LIN {X 0,Y 612.539,Z 280.742,A -85,B 0,C 180,E1 -8059.322,E2 -8059.322} C_VEL
LIN {X 0,Y 612.53,Z 280.74,A -85,B 0,C 180,E1 -8062.097,E2 -8062.097} C_VEL
LIN {X 0,Y 612.605,Z 280.734,A -85,B 0,C 180,E1 -8064.329,E2 -8064.329} C_VEL
LIN {X 0,Y 612.556,Z 280.744,A -85,B 0,C 180,E1 -8066.71,E2 -8066.71} C_VEL
LIN {X 0,Y 612.575,Z 280.737,A -85,B 0,C 180,E1 -8069.048,E2 -8069.048} C_VEL
LIN {X 0,Y 612.575,Z 280.734,A -85,B 0,C 180,E1 -8071.698,E2 -8071.698} C_VEL
LIN {X 0,Y 612.557,Z 280.743,A -85,B 0,C 180,E1 -8074.603,E2 -8074.603} C_VEL
LIN {X 0,Y 612.586,Z 280.736,A -85,B 0,C 180,E1 -8077.122,E2 -8077.122} C_VEL
LIN {X 0,Y 612.607,Z 280.742,A -85,B 0,C 180,E1 -8079.939,E2 -8079.939} C_VEL
LIN {X 0,Y 612.586,Z 280.735,A -85,B 0,C 180,E1 -8082.705,E2 -8082.705} C_VEL
LIN {X 0,Y 612.61,Z 280.735,A -85,B 0,C 180,E1 -8085.431,E2 -8085.431} C_VEL
LIN {X 0,Y 612.595,Z 280.739,A -85,B 0,C 180,E1 -8087.453,E2 -8087.453} C_VEL
LIN {X 0,Y 612.647,Z 280.829,A -85,B 0,C 180,E1 -8088.751,E2 -8088.751} C_VEL
LIN {X 0,Y 614.455,Z 290.422,A -85,B 0,C 180,E1 -8089.989,E2 -8089.989} C_VEL
LIN {X 0,Y 614.314,Z 310.578,A -85,B 0,C 180,E1 -8092.465,E2 -8092.465} C_VEL
LIN {X 0,Y 613.746,Z 335.947,A -85,B 0,C 180,E1 -8095.582,E2 -8095.582} C_VEL
LIN {X 0,Y 613.659,Z 342.221,A -85,B 0,C 180,E1 -8096.36,E2 -8096.36} C_VEL
LIN {X 0,Y 616.099,Z 357.034,A -85,B 0,C 180,E1 -8096.639,E2 -8096.639} C_VEL
LIN {X 0,Y 614.848,Z 480.497,A -85,B 0,C 180,E1 -8098.246,E2 -8098.246} C_VEL
LIN {X 0,Y 614.62,Z 495.222,A -85,B 0,C 180,E1 -8098.571,E2 -8098.571} C_VEL
LIN {X 0,Y 614.253,Z 509.138,A -85,B 0,C 180,E1 -8099.02,E2 -8099.02} C_VEL
LIN {X 0,Y 613.913,Z 520.829,A -85,B 0,C 180,E1 -8099.51,E2 -8099.51} C_VEL
LIN {X 0,Y 613.489,Z 533.262,A -85,B 0,C 180,E1 -8100.164,E2 -8100.164} C_VEL
LIN {X 0,Y 613.212,Z 545.749,A -85,B 0,C 180,E1 -8100.982,E2 -8100.982} C_VEL
LIN {X 0,Y 612.816,Z 556.08,A -85,B 0,C 180,E1 -8101.801,E2 -8101.801} C_VEL
LIN {X 0,Y 612.393,Z 566.382,A -85,B 0,C 180,E1 -8102.786,E2 -8102.786} C_VEL
LIN {X 0,Y 612.12,Z 574.899,A -85,B 0,C 180,E1 -8103.773,E2 -8103.773} C_VEL
LIN {X 0,Y 611.915,Z 583.24,A -85,B 0,C 180,E1 -8104.95,E2 -8104.95} C_VEL
LIN {X 0,Y 611.86,Z 588.773,A -85,B 0,C 180,E1 -8105.914,E2 -8105.914} C_VEL
LIN {X 0,Y 611.734,Z 593.465,A -85,B 0,C 180,E1 -8106.905,E2 -8106.905} C_VEL
LIN {X 0,Y 611.594,Z 598.317,A -85,B 0,C 180,E1 -8108.231,E2 -8108.231} C_VEL
LIN {X 0,Y 611.56,Z 600.925,A -85,B 0,C 180,E1 -8109.227,E2 -8109.227} C_VEL
LIN {X 0,Y 611.605,Z 602.329,A -85,B 0,C 180,E1 -8109.959,E2 -8109.959} C_VEL
LIN {X 0,Y 611.466,Z 603.754,A -85,B 0,C 180,E1 -8111.229,E2 -8111.229} C_VEL
LIN {X 0,Y 611.5,Z 603.889,A -85,B 0,C 180,E1 -8112.57,E2 -8112.57} C_VEL
LIN {X 0,Y 611.564,Z 603.427,A -85,B 0,C 180,E1 -8113.242,E2 -8113.242} C_VEL
LIN {X 0,Y 611.514,Z 601.388,A -85,B 0,C 180,E1 -8114.596,E2 -8114.596} C_VEL
LIN {X 0,Y 611.62,Z 597.836,A -85,B 0,C 180,E1 -8115.953,E2 -8115.953} C_VEL
LIN {X 0,Y 611.67,Z 594.126,A -85,B 0,C 180,E1 -8116.978,E2 -8116.978} C_VEL
LIN {X 0,Y 611.798,Z 588.668,A -85,B 0,C 180,E1 -8118.144,E2 -8118.144} C_VEL
LIN {X 0,Y 611.995,Z 581.268,A -85,B 0,C 180,E1 -8119.385,E2 -8119.385} C_VEL
LIN {X 0,Y 612.218,Z 573.296,A -85,B 0,C 180,E1 -8120.464,E2 -8120.464} C_VEL
LIN {X 0,Y 612.47,Z 564.315,A -85,B 0,C 180,E1 -8121.467,E2 -8121.467} C_VEL
LIN {X 0,Y 612.872,Z 553.36,A -85,B 0,C 180,E1 -8122.476,E2 -8122.476} C_VEL
LIN {X 0,Y 613.238,Z 542.494,A -85,B 0,C 180,E1 -8123.296,E2 -8123.296} C_VEL
LIN {X 0,Y 613.619,Z 530.354,A -85,B 0,C 180,E1 -8124.047,E2 -8124.047} C_VEL
LIN {X 0,Y 613.943,Z 517.245,A -85,B 0,C 180,E1 -8124.699,E2 -8124.699} C_VEL
LIN {X 0,Y 614.354,Z 503.666,A -85,B 0,C 180,E1 -8125.222,E2 -8125.222} C_VEL
LIN {X 0,Y 614.635,Z 489.847,A -85,B 0,C 180,E1 -8125.616,E2 -8125.616} C_VEL
LIN {X 0,Y 614.816,Z 476.132,A -85,B 0,C 180,E1 -8125.88,E2 -8125.88} C_VEL
LIN {X 0,Y 615.787,Z 356.431,A -85,B 0,C 180,E1 -8127.383,E2 -8127.383} C_VEL
LIN {X 0,Y 613.434,Z 341.628,A -85,B 0,C 180,E1 -8127.642,E2 -8127.642} C_VEL
LIN {X 0,Y 613.881,Z 320.293,A -85,B 0,C 180,E1 -8130.325,E2 -8130.325} C_VEL
LIN {X 0,Y 614.329,Z 299.291,A -85,B 0,C 180,E1 -8132.967,E2 -8132.967} C_VEL
LIN {X 0,Y 614.456,Z 291.433,A -85,B 0,C 180,E1 -8133.957,E2 -8133.957} C_VEL
LIN {X 0,Y 612.592,Z 280.737,A -85,B 0,C 180,E1 -8135.395,E2 -8135.395} C_VEL
LIN {X 0,Y 612.548,Z 280.745,A -85,B 0,C 180,E1 -8138.133,E2 -8138.133} C_VEL
LIN {X 0,Y 612.54,Z 280.738,A -85,B 0,C 180,E1 -8140.998,E2 -8140.998} C_VEL
LIN {X 0,Y 612.553,Z 280.742,A -85,B 0,C 180,E1 -8143.912,E2 -8143.912} C_VEL
LIN {X 0,Y 612.551,Z 280.743,A -85,B 0,C 180,E1 -8144.184,E2 -8144.184} C_VEL
LIN {X 0,Y 611.899,Z 280.825,A -85,B 0,C 180,E1 -8144.733,E2 -8144.733} C_VEL
LIN {X 0,Y 609.053,Z 281.178,A -85,B 0,C 180,E1 -8145.624,E2 -8145.624} C_VEL
LIN {X 0,Y 606.631,Z 281.478,A -85,B 0,C 180,E1 -8146.34,E2 -8146.34} C_VEL
LIN {X 0,Y 605.577,Z 281.607,A -85,B 0,C 180,E1 -8146.893,E2 -8146.893} C_VEL
LIN {X 0,Y 605.485,Z 281.618,A -85,B 0,C 180,E1 -8147.08,E2 -8147.08} C_VEL
LIN {X 0,Y 605.499,Z 281.622,A -85,B 0,C 180,E1 -8149.773,E2 -8149.773} C_VEL
LIN {X 0,Y 605.482,Z 281.62,A -85,B 0,C 180,E1 -8152.183,E2 -8152.183} C_VEL
LIN {X 0,Y 605.512,Z 281.616,A -85,B 0,C 180,E1 -8154.661,E2 -8154.661} C_VEL
LIN {X 0,Y 605.519,Z 281.619,A -85,B 0,C 180,E1 -8157.612,E2 -8157.612} C_VEL
LIN {X 0,Y 605.509,Z 281.616,A -85,B 0,C 180,E1 -8160.18,E2 -8160.18} C_VEL
LIN {X 0,Y 605.497,Z 281.62,A -85,B 0,C 180,E1 -8162.436,E2 -8162.436} C_VEL
LIN {X 0,Y 605.528,Z 281.615,A -85,B 0,C 180,E1 -8165.389,E2 -8165.389} C_VEL
LIN {X 0,Y 605.548,Z 281.615,A -85,B 0,C 180,E1 -8168.274,E2 -8168.274} C_VEL
LIN {X 0,Y 605.564,Z 281.61,A -85,B 0,C 180,E1 -8171.101,E2 -8171.101} C_VEL
LIN {X 0,Y 605.58,Z 281.609,A -85,B 0,C 180,E1 -8173.882,E2 -8173.882} C_VEL
LIN {X 0,Y 605.61,Z 281.604,A -85,B 0,C 180,E1 -8176.624,E2 -8176.624} C_VEL
LIN {X 0,Y 605.595,Z 281.605,A -85,B 0,C 180,E1 -8179.46,E2 -8179.46} C_VEL
LIN {X 0,Y 605.638,Z 281.602,A -85,B 0,C 180,E1 -8182.69,E2 -8182.69} C_VEL
LIN {X 0,Y 605.665,Z 281.693,A -85,B 0,C 180,E1 -8183.534,E2 -8183.534} C_VEL
LIN {X 0,Y 606.536,Z 288.286,A -85,B 0,C 180,E1 -8184.698,E2 -8184.698} C_VEL
LIN {X 0,Y 606.366,Z 297.794,A -85,B 0,C 180,E1 -8186.314,E2 -8186.314} C_VEL
LIN {X 0,Y 609.016,Z 310.551,A -85,B 0,C 180,E1 -8186.537,E2 -8186.537} C_VEL
LIN {X 0,Y 608.253,Z 432.958,A -85,B 0,C 180,E1 -8187.998,E2 -8187.998} C_VEL
LIN {X 0,Y 608.073,Z 447.42,A -85,B 0,C 180,E1 -8188.307,E2 -8188.307} C_VEL
LIN {X 0,Y 607.806,Z 460.691,A -85,B 0,C 180,E1 -8188.719,E2 -8188.719} C_VEL
LIN {X 0,Y 607.447,Z 473.678,A -85,B 0,C 180,E1 -8189.255,E2 -8189.255} C_VEL
LIN {X 0,Y 607.1,Z 486.217,A -85,B 0,C 180,E1 -8189.916,E2 -8189.916} C_VEL
LIN {X 0,Y 606.605,Z 497.697,A -85,B 0,C 180,E1 -8190.66,E2 -8190.66} C_VEL
LIN {X 0,Y 606.277,Z 508.19,A -85,B 0,C 180,E1 -8191.488,E2 -8191.488} C_VEL
LIN {X 0,Y 605.795,Z 518.648,A -85,B 0,C 180,E1 -8192.483,E2 -8192.483} C_VEL
LIN {X 0,Y 605.512,Z 527.271,A -85,B 0,C 180,E1 -8193.48,E2 -8193.48} C_VEL
LIN {X 0,Y 605.174,Z 534.48,A -85,B 0,C 180,E1 -8194.479,E2 -8194.479} C_VEL
LIN {X 0,Y 605.072,Z 541.182,A -85,B 0,C 180,E1 -8195.612,E2 -8195.612} C_VEL
LIN {X 0,Y 604.868,Z 546.167,A -85,B 0,C 180,E1 -8196.648,E2 -8196.648} C_VEL
LIN {X 0,Y 604.685,Z 551.137,A -85,B 0,C 180,E1 -8197.988,E2 -8197.988} C_VEL
LIN {X 0,Y 604.615,Z 554.619,A -85,B 0,C 180,E1 -8199.332,E2 -8199.332} C_VEL
LIN {X 0,Y 604.562,Z 556.716,A -85,B 0,C 180,E1 -8200.681,E2 -8200.681} C_VEL
LIN {X 0,Y 604.528,Z 557.462,A -85,B 0,C 180,E1 -8202.036,E2 -8202.036} C_VEL
LIN {X 0,Y 604.611,Z 556.839,A -85,B 0,C 180,E1 -8203.395,E2 -8203.395} C_VEL
LIN {X 0,Y 604.618,Z 554.819,A -85,B 0,C 180,E1 -8204.764,E2 -8204.764} C_VEL
LIN {X 0,Y 604.762,Z 551.338,A -85,B 0,C 180,E1 -8206.137,E2 -8206.137} C_VEL
LIN {X 0,Y 604.901,Z 546.275,A -85,B 0,C 180,E1 -8207.52,E2 -8207.52} C_VEL
LIN {X 0,Y 605.11,Z 541.411,A -85,B 0,C 180,E1 -8208.541,E2 -8208.541} C_VEL
LIN {X 0,Y 605.398,Z 534.08,A -85,B 0,C 180,E1 -8209.779,E2 -8209.779} C_VEL
LIN {X 0,Y 605.675,Z 526.294,A -85,B 0,C 180,E1 -8210.845,E2 -8210.845} C_VEL
LIN {X 0,Y 606.124,Z 517.12,A -85,B 0,C 180,E1 -8211.879,E2 -8211.879} C_VEL
LIN {X 0,Y 606.513,Z 507.043,A -85,B 0,C 180,E1 -8212.821,E2 -8212.821} C_VEL
LIN {X 0,Y 607.008,Z 495.237,A -85,B 0,C 180,E1 -8213.728,E2 -8213.728} C_VEL
LIN {X 0,Y 607.408,Z 483.868,A -85,B 0,C 180,E1 -8214.44,E2 -8214.44} C_VEL
LIN {X 0,Y 607.866,Z 470.729,A -85,B 0,C 180,E1 -8215.097,E2 -8215.097} C_VEL
LIN {X 0,Y 608.202,Z 456.909,A -85,B 0,C 180,E1 -8215.63,E2 -8215.63} C_VEL
LIN {X 0,Y 608.475,Z 441.955,A -85,B 0,C 180,E1 -8216.045,E2 -8216.045} C_VEL
LIN {X 0,Y 608.6,Z 428.129,A -85,B 0,C 180,E1 -8216.291,E2 -8216.291} C_VEL
LIN {X 0,Y 609.415,Z 310.991,A -85,B 0,C 180,E1 -8217.691,E2 -8217.691} C_VEL
LIN {X 0,Y 606.657,Z 298.091,A -85,B 0,C 180,E1 -8217.943,E2 -8217.943} C_VEL
LIN {X 0,Y 606.757,Z 288.755,A -85,B 0,C 180,E1 -8219.569,E2 -8219.569} C_VEL
LIN {X 0,Y 605.499,Z 281.623,A -85,B 0,C 180,E1 -8220.897,E2 -8220.897} C_VEL
LIN {X 0,Y 605.495,Z 281.62,A -85,B 0,C 180,E1 -8223.727,E2 -8223.727} C_VEL
LIN {X 0,Y 605.501,Z 281.623,A -85,B 0,C 180,E1 -8226.152,E2 -8226.152} C_VEL
LIN {X 0,Y 605.486,Z 281.616,A -85,B 0,C 180,E1 -8229.188,E2 -8229.188} C_VEL
LIN {X 0,Y 605.471,Z 281.624,A -85,B 0,C 180,E1 -8232.14,E2 -8232.14} C_VEL
LIN {X 0,Y 605.489,Z 281.609,A -85,B 0,C 180,E1 -8234.88,E2 -8234.88} C_VEL
LIN {X 0,Y 605.48,Z 281.624,A -85,B 0,C 180,E1 -8237.858,E2 -8237.858} C_VEL
LIN {X 0,Y 605.487,Z 281.617,A -85,B 0,C 180,E1 -8240.487,E2 -8240.487} C_VEL
LIN {X 0,Y 605.524,Z 281.609,A -85,B 0,C 180,E1 -8243.022,E2 -8243.022} C_VEL
LIN {X 0,Y 605.481,Z 281.611,A -85,B 0,C 180,E1 -8245.469,E2 -8245.469} C_VEL
LIN {X 0,Y 605.492,Z 281.622,A -85,B 0,C 180,E1 -8247.85,E2 -8247.85} C_VEL
LIN {X 0,Y 605.528,Z 281.614,A -85,B 0,C 180,E1 -8250.172,E2 -8250.172} C_VEL
LIN {X 0,Y 605.487,Z 281.612,A -85,B 0,C 180,E1 -8252.437,E2 -8252.437} C_VEL
LIN {X 0,Y 605.509,Z 281.62,A -85,B 0,C 180,E1 -8255.39,E2 -8255.39} C_VEL
LIN {X 0,Y 605.53,Z 281.618,A -85,B 0,C 180,E1 -8257.722,E2 -8257.722} C_VEL
LIN {X 0,Y 605.527,Z 281.608,A -85,B 0,C 180,E1 -8260.4,E2 -8260.4} C_VEL
LIN {X 0,Y 605.517,Z 281.617,A -85,B 0,C 180,E1 -8263.19,E2 -8263.19} C_VEL
LIN {X 0,Y 605.567,Z 281.603,A -85,B 0,C 180,E1 -8265.942,E2 -8265.942} C_VEL
LIN {X 0,Y 605.545,Z 281.609,A -85,B 0,C 180,E1 -8268.659,E2 -8268.659} C_VEL
LIN {X 0,Y 605.533,Z 281.608,A -85,B 0,C 180,E1 -8270.68,E2 -8270.68} C_VEL
LIN {X 0,Y 605.638,Z 281.605,A -85,B 0,C 180,E1 -8273.359,E2 -8273.359} C_VEL
LIN {X 0,Y 605.651,Z 281.589,A -85,B 0,C 180,E1 -8276.021,E2 -8276.021} C_VEL
LIN {X 0,Y 605.776,Z 281.585,A -85,B 0,C 180,E1 -8279.338,E2 -8279.338} C_VEL
LIN {X 0,Y 605.781,Z 281.578,A -85,B 0,C 180,E1 -8281.325,E2 -8281.325} C_VEL
LIN {X 0,Y 605.666,Z 281.597,A -85,B 0,C 180,E1 -8284.643,E2 -8284.643} C_VEL
LIN {X 0,Y 605.616,Z 281.598,A -85,B 0,C 180,E1 -8287.309,E2 -8287.309} C_VEL
LIN {X 0,Y 605.635,Z 281.602,A -85,B 0,C 180,E1 -8290.664,E2 -8290.664} C_VEL
LIN {X 0,Y 605.588,Z 281.6,A -85,B 0,C 180,E1 -8293.705,E2 -8293.705} C_VEL
LIN {X 0,Y 605.543,Z 281.611,A -85,B 0,C 180,E1 -8296.809,E2 -8296.809} C_VEL
LIN {X 0,Y 605.543,Z 281.615,A -85,B 0,C 180,E1 -8298.898,E2 -8298.898} C_VEL
LIN {X 0,Y 605.519,Z 281.607,A -85,B 0,C 180,E1 -8301.726,E2 -8301.726} C_VEL
LIN {X 0,Y 605.523,Z 281.611,A -85,B 0,C 180,E1 -8303.965,E2 -8303.965} C_VEL
LIN {X 0,Y 605.476,Z 281.622,A -85,B 0,C 180,E1 -8306.819,E2 -8306.819} C_VEL
LIN {X 0,Y 605.529,Z 281.612,A -85,B 0,C 180,E1 -8309.067,E2 -8309.067} C_VEL
LIN {X 0,Y 605.536,Z 281.609,A -85,B 0,C 180,E1 -8311.368,E2 -8311.368} C_VEL
LIN {X 0,Y 605.514,Z 281.608,A -85,B 0,C 180,E1 -8314.529,E2 -8314.529} C_VEL
LIN {X 0,Y 605.549,Z 281.606,A -85,B 0,C 180,E1 -8317.052,E2 -8317.052} C_VEL
LIN {X 0,Y 605.509,Z 281.613,A -85,B 0,C 180,E1 -8319.512,E2 -8319.512} C_VEL
LIN {X 0,Y 605.507,Z 281.621,A -85,B 0,C 180,E1 -8322.243,E2 -8322.243} C_VEL
LIN {X 0,Y 605.499,Z 281.613,A -85,B 0,C 180,E1 -8325.121,E2 -8325.121} C_VEL
LIN {X 0,Y 605.53,Z 281.615,A -85,B 0,C 180,E1 -8327.866,E2 -8327.866} C_VEL
LIN {X 0,Y 605.514,Z 281.617,A -85,B 0,C 180,E1 -8330.492,E2 -8330.492} C_VEL
LIN {X 0,Y 605.581,Z 281.604,A -85,B 0,C 180,E1 -8333.028,E2 -8333.028} C_VEL
LIN {X 0,Y 605.519,Z 281.619,A -85,B 0,C 180,E1 -8335.474,E2 -8335.474} C_VEL
LIN {X 0,Y 605.51,Z 281.626,A -85,B 0,C 180,E1 -8337.854,E2 -8337.854} C_VEL
LIN {X 0,Y 605.54,Z 281.619,A -85,B 0,C 180,E1 -8340.175,E2 -8340.175} C_VEL
LIN {X 0,Y 605.504,Z 281.62,A -85,B 0,C 180,E1 -8342.44,E2 -8342.44} C_VEL
LIN {X 0,Y 605.53,Z 281.746,A -85,B 0,C 180,E1 -8343.857,E2 -8343.857} C_VEL
LIN {X 0,Y 608.272,Z 294.613,A -85,B 0,C 180,E1 -8345.629,E2 -8345.629} C_VEL
LIN {X 0,Y 608.596,Z 297.957,A -85,B 0,C 180,E1 -8346.067,E2 -8346.067} C_VEL
LIN {X 0,Y 607.542,Z 322.009,A -85,B 0,C 180,E1 -8349.045,E2 -8349.045} C_VEL
LIN {X 0,Y 606.776,Z 343.571,A -85,B 0,C 180,E1 -8351.67,E2 -8351.67} C_VEL
LIN {X 0,Y 606.202,Z 363.615,A -85,B 0,C 180,E1 -8354.085,E2 -8354.085} C_VEL
LIN {X 0,Y 609.134,Z 386.789,A -85,B 0,C 180,E1 -8354.452,E2 -8354.452} C_VEL
LIN {X 0,Y 608.328,Z 501.983,A -85,B 0,C 180,E1 -8355.839,E2 -8355.839} C_VEL
LIN {X 0,Y 607.944,Z 516.52,A -85,B 0,C 180,E1 -8356.149,E2 -8356.149} C_VEL
LIN {X 0,Y 607.509,Z 530.447,A -85,B 0,C 180,E1 -8356.585,E2 -8356.585} C_VEL
LIN {X 0,Y 607.014,Z 544.312,A -85,B 0,C 180,E1 -8357.168,E2 -8357.168} C_VEL
LIN {X 0,Y 606.511,Z 556.746,A -85,B 0,C 180,E1 -8357.835,E2 -8357.835} C_VEL
LIN {X 0,Y 606.021,Z 569.306,A -85,B 0,C 180,E1 -8358.67,E2 -8358.67} C_VEL
LIN {X 0,Y 605.703,Z 580.12,A -85,B 0,C 180,E1 -8359.553,E2 -8359.553} C_VEL
LIN {X 0,Y 605.319,Z 589.873,A -85,B 0,C 180,E1 -8360.511,E2 -8360.511} C_VEL
LIN {X 0,Y 604.947,Z 598.392,A -85,B 0,C 180,E1 -8361.512,E2 -8361.512} C_VEL
LIN {X 0,Y 604.739,Z 606.555,A -85,B 0,C 180,E1 -8362.682,E2 -8362.682} C_VEL
LIN {X 0,Y 604.599,Z 614.233,A -85,B 0,C 180,E1 -8364.017,E2 -8364.017} C_VEL
LIN {X 0,Y 604.55,Z 620.167,A -85,B 0,C 180,E1 -8365.35,E2 -8365.35} C_VEL
LIN {X 0,Y 604.531,Z 624.481,A -85,B 0,C 180,E1 -8366.681,E2 -8366.681} C_VEL
LIN {X 0,Y 604.515,Z 627.303,A -85,B 0,C 180,E1 -8368.01,E2 -8368.01} C_VEL
LIN {X 0,Y 604.578,Z 628.713,A -85,B 0,C 180,E1 -8369.338,E2 -8369.338} C_VEL
LIN {X 0,Y 604.567,Z 628.72,A -85,B 0,C 180,E1 -8370.665,E2 -8370.665} C_VEL
LIN {X 0,Y 604.516,Z 627.318,A -85,B 0,C 180,E1 -8371.994,E2 -8371.994} C_VEL
LIN {X 0,Y 604.531,Z 624.497,A -85,B 0,C 180,E1 -8373.323,E2 -8373.323} C_VEL
LIN {X 0,Y 604.553,Z 620.183,A -85,B 0,C 180,E1 -8374.654,E2 -8374.654} C_VEL
LIN {X 0,Y 604.601,Z 614.25,A -85,B 0,C 180,E1 -8375.986,E2 -8375.986} C_VEL
LIN {X 0,Y 604.717,Z 607.53,A -85,B 0,C 180,E1 -8377.154,E2 -8377.154} C_VEL
LIN {X 0,Y 604.937,Z 597.942,A -85,B 0,C 180,E1 -8378.491,E2 -8378.491} C_VEL
LIN {X 0,Y 605.238,Z 589.299,A -85,B 0,C 180,E1 -8379.494,E2 -8379.494} C_VEL
LIN {X 0,Y 605.643,Z 579.617,A -85,B 0,C 180,E1 -8380.427,E2 -8380.427} C_VEL
LIN {X 0,Y 605.993,Z 568.254,A -85,B 0,C 180,E1 -8381.334,E2 -8381.334} C_VEL
LIN {X 0,Y 606.38,Z 556.766,A -85,B 0,C 180,E1 -8382.087,E2 -8382.087} C_VEL
LIN {X 0,Y 606.861,Z 544.201,A -85,B 0,C 180,E1 -8382.754,E2 -8382.754} C_VEL
LIN {X 0,Y 607.302,Z 530.148,A -85,B 0,C 180,E1 -8383.338,E2 -8383.338} C_VEL
LIN {X 0,Y 607.747,Z 515.928,A -85,B 0,C 180,E1 -8383.774,E2 -8383.774} C_VEL
LIN {X 0,Y 608.063,Z 502.106,A -85,B 0,C 180,E1 -8384.062,E2 -8384.062} C_VEL
LIN {X 0,Y 608.721,Z 384.956,A -85,B 0,C 180,E1 -8385.46,E2 -8385.46} C_VEL
LIN {X 0,Y 606.082,Z 363.877,A -85,B 0,C 180,E1 -8385.782,E2 -8385.782} C_VEL
LIN {X 0,Y 606.757,Z 337.997,A -85,B 0,C 180,E1 -8388.86,E2 -8388.86} C_VEL
LIN {X 0,Y 607.532,Z 314.727,A -85,B 0,C 180,E1 -8391.652,E2 -8391.652} C_VEL
LIN {X 0,Y 608.246,Z 295.852,A -85,B 0,C 180,E1 -8393.941,E2 -8393.941} C_VEL
LIN {X 0,Y 605.821,Z 283.126,A -85,B 0,C 180,E1 -8395.6,E2 -8395.6} C_VEL
LIN {X 0,Y 605.521,Z 281.62,A -85,B 0,C 180,E1 -8395.828,E2 -8395.828} C_VEL
LIN {X 0,Y 605.535,Z 281.614,A -85,B 0,C 180,E1 -8398.464,E2 -8398.464} C_VEL
LIN {X 0,Y 605.508,Z 281.618,A -85,B 0,C 180,E1 -8401.371,E2 -8401.371} C_VEL
LIN {X 0,Y 605.513,Z 281.622,A -85,B 0,C 180,E1 -8403.73,E2 -8403.73} C_VEL
LIN {X 0,Y 605.509,Z 281.617,A -85,B 0,C 180,E1 -8406.156,E2 -8406.156} C_VEL
LIN {X 0,Y 605.504,Z 281.621,A -85,B 0,C 180,E1 -8409.19,E2 -8409.19} C_VEL
LIN {X 0,Y 605.484,Z 281.616,A -85,B 0,C 180,E1 -8412.143,E2 -8412.143} C_VEL
LIN {X 0,Y 605.506,Z 281.621,A -85,B 0,C 180,E1 -8415.118,E2 -8415.118} C_VEL
LIN {X 0,Y 605.485,Z 281.617,A -85,B 0,C 180,E1 -8417.858,E2 -8417.858} C_VEL
LIN {X 0,Y 605.505,Z 281.622,A -85,B 0,C 180,E1 -8420.811,E2 -8420.811} C_VEL
LIN {X 0,Y 605.565,Z 281.608,A -85,B 0,C 180,E1 -8424.066,E2 -8424.066} C_VEL
LIN {X 0,Y 605.499,Z 281.619,A -85,B 0,C 180,E1 -8427.064,E2 -8427.064} C_VEL
LIN {X 0,Y 605.518,Z 281.614,A -85,B 0,C 180,E1 -8429.404,E2 -8429.404} C_VEL
LIN {X 0,Y 605.536,Z 281.611,A -85,B 0,C 180,E1 -8431.689,E2 -8431.689} C_VEL
LIN {X 0,Y 605.52,Z 281.619,A -85,B 0,C 180,E1 -8434.659,E2 -8434.659} C_VEL
LIN {X 0,Y 605.544,Z 281.614,A -85,B 0,C 180,E1 -8436.841,E2 -8436.841} C_VEL
LIN {X 0,Y 605.564,Z 281.616,A -85,B 0,C 180,E1 -8439.696,E2 -8439.696} C_VEL
LIN {X 0,Y 605.55,Z 281.614,A -85,B 0,C 180,E1 -8442.498,E2 -8442.498} C_VEL
LIN {X 0,Y 605.555,Z 281.613,A -85,B 0,C 180,E1 -8445.258,E2 -8445.258} C_VEL
LIN {X 0,Y 605.554,Z 281.615,A -85,B 0,C 180,E1 -8447.304,E2 -8447.304} C_VEL
LIN {X 0,Y 605.61,Z 281.71,A -85,B 0,C 180,E1 -8448.576,E2 -8448.576} C_VEL
LIN {X 0,Y 607.526,Z 291.601,A -85,B 0,C 180,E1 -8449.873,E2 -8449.873} C_VEL
LIN {X 0,Y 607.39,Z 310.649,A -85,B 0,C 180,E1 -8452.229,E2 -8452.229} C_VEL
LIN {X 0,Y 606.829,Z 333.374,A -85,B 0,C 180,E1 -8455.034,E2 -8455.034} C_VEL
LIN {X 0,Y 606.742,Z 342.632,A -85,B 0,C 180,E1 -8456.163,E2 -8456.163} C_VEL
LIN {X 0,Y 609.311,Z 358.124,A -85,B 0,C 180,E1 -8456.457,E2 -8456.457} C_VEL
LIN {X 0,Y 607.981,Z 480.382,A -85,B 0,C 180,E1 -8458.081,E2 -8458.081} C_VEL
LIN {X 0,Y 607.746,Z 494.392,A -85,B 0,C 180,E1 -8458.39,E2 -8458.39} C_VEL
LIN {X 0,Y 607.347,Z 508.656,A -85,B 0,C 180,E1 -8458.844,E2 -8458.844} C_VEL
LIN {X 0,Y 607.014,Z 520.456,A -85,B 0,C 180,E1 -8459.339,E2 -8459.339} C_VEL
LIN {X 0,Y 606.567,Z 533.003,A -85,B 0,C 180,E1 -8460,E2 -8460} C_VEL
LIN {X 0,Y 606.237,Z 545.558,A -85,B 0,C 180,E1 -8460.827,E2 -8460.827} C_VEL
LIN {X 0,Y 605.829,Z 555.939,A -85,B 0,C 180,E1 -8461.656,E2 -8461.656} C_VEL
LIN {X 0,Y 605.368,Z 566.288,A -85,B 0,C 180,E1 -8462.653,E2 -8462.653} C_VEL
LIN {X 0,Y 605.122,Z 574.839,A -85,B 0,C 180,E1 -8463.65,E2 -8463.65} C_VEL
LIN {X 0,Y 604.97,Z 581.966,A -85,B 0,C 180,E1 -8464.649,E2 -8464.649} C_VEL
LIN {X 0,Y 604.807,Z 588.518,A -85,B 0,C 180,E1 -8465.765,E2 -8465.765} C_VEL
LIN {X 0,Y 604.628,Z 594.233,A -85,B 0,C 180,E1 -8466.987,E2 -8466.987} C_VEL
LIN {X 0,Y 604.506,Z 597.869,A -85,B 0,C 180,E1 -8467.993,E2 -8467.993} C_VEL
LIN {X 0,Y 604.484,Z 601.393,A -85,B 0,C 180,E1 -8469.336,E2 -8469.336} C_VEL
LIN {X 0,Y 604.431,Z 603.486,A -85,B 0,C 180,E1 -8470.685,E2 -8470.685} C_VEL
LIN {X 0,Y 604.39,Z 604.167,A -85,B 0,C 180,E1 -8472.041,E2 -8472.041} C_VEL
LIN {X 0,Y 604.465,Z 603.4,A -85,B 0,C 180,E1 -8473.401,E2 -8473.401} C_VEL
LIN {X 0,Y 604.424,Z 601.187,A -85,B 0,C 180,E1 -8474.771,E2 -8474.771} C_VEL
LIN {X 0,Y 604.544,Z 597.466,A -85,B 0,C 180,E1 -8476.145,E2 -8476.145} C_VEL
LIN {X 0,Y 604.607,Z 593.577,A -85,B 0,C 180,E1 -8477.183,E2 -8477.183} C_VEL
LIN {X 0,Y 604.731,Z 588.628,A -85,B 0,C 180,E1 -8478.232,E2 -8478.232} C_VEL
LIN {X 0,Y 604.927,Z 581.455,A -85,B 0,C 180,E1 -8479.445,E2 -8479.445} C_VEL
LIN {X 0,Y 605.152,Z 573.949,A -85,B 0,C 180,E1 -8480.478,E2 -8480.478} C_VEL
LIN {X 0,Y 605.448,Z 564.502,A -85,B 0,C 180,E1 -8481.55,E2 -8481.55} C_VEL
LIN {X 0,Y 605.826,Z 554.145,A -85,B 0,C 180,E1 -8482.519,E2 -8482.519} C_VEL
LIN {X 0,Y 606.222,Z 542.664,A -85,B 0,C 180,E1 -8483.402,E2 -8483.402} C_VEL
LIN {X 0,Y 606.65,Z 529.898,A -85,B 0,C 180,E1 -8484.195,E2 -8484.195} C_VEL
LIN {X 0,Y 606.964,Z 517.413,A -85,B 0,C 180,E1 -8484.82,E2 -8484.82} C_VEL
LIN {X 0,Y 607.397,Z 503.849,A -85,B 0,C 180,E1 -8485.348,E2 -8485.348} C_VEL
LIN {X 0,Y 607.696,Z 490.067,A -85,B 0,C 180,E1 -8485.747,E2 -8485.747} C_VEL
LIN {X 0,Y 607.901,Z 475.357,A -85,B 0,C 180,E1 -8486.03,E2 -8486.03} C_VEL
LIN {X 0,Y 608.819,Z 356.567,A -85,B 0,C 180,E1 -8487.549,E2 -8487.549} C_VEL
LIN {X 0,Y 606.453,Z 341.695,A -85,B 0,C 180,E1 -8487.816,E2 -8487.816} C_VEL
LIN {X 0,Y 606.91,Z 321.45,A -85,B 0,C 180,E1 -8490.377,E2 -8490.377} C_VEL
LIN {X 0,Y 607.475,Z 297.497,A -85,B 0,C 180,E1 -8493.407,E2 -8493.407} C_VEL
LIN {X 0,Y 607.274,Z 290.841,A -85,B 0,C 180,E1 -8494.267,E2 -8494.267} C_VEL
LIN {X 0,Y 605.566,Z 281.613,A -85,B 0,C 180,E1 -8495.511,E2 -8495.511} C_VEL
LIN {X 0,Y 605.511,Z 281.621,A -85,B 0,C 180,E1 -8498.129,E2 -8498.129} C_VEL
LIN {X 0,Y 605.502,Z 281.621,A -85,B 0,C 180,E1 -8500.376,E2 -8500.376} C_VEL
LIN {X 0,Y 605.515,Z 281.614,A -85,B 0,C 180,E1 -8503.215,E2 -8503.215} C_VEL
LIN {X 0,Y 605.505,Z 281.622,A -85,B 0,C 180,E1 -8506.045,E2 -8506.045} C_VEL
LIN {X 0,Y 605.485,Z 281.618,A -85,B 0,C 180,E1 -8507.08,E2 -8507.08} C_VEL
LIN {X 0,Y 604.806,Z 281.707,A -85,B 0,C 180,E1 -8507.636,E2 -8507.636} C_VEL
LIN {X 0,Y 601.966,Z 282.064,A -85,B 0,C 180,E1 -8508.538,E2 -8508.538} C_VEL
LIN {X 0,Y 599.573,Z 282.364,A -85,B 0,C 180,E1 -8509.263,E2 -8509.263} C_VEL
LIN {X 0,Y 598.541,Z 282.49,A -85,B 0,C 180,E1 -8509.822,E2 -8509.822} C_VEL
LIN {X 0,Y 598.454,Z 282.499,A -85,B 0,C 180,E1 -8510.012,E2 -8510.012} C_VEL
LIN {X 0,Y 598.44,Z 282.497,A -85,B 0,C 180,E1 -8512.741,E2 -8512.741} C_VEL
LIN {X 0,Y 598.463,Z 282.496,A -85,B 0,C 180,E1 -8515.013,E2 -8515.013} C_VEL
LIN {X 0,Y 598.466,Z 282.496,A -85,B 0,C 180,E1 -8517.425,E2 -8517.425} C_VEL
LIN {X 0,Y 598.463,Z 282.494,A -85,B 0,C 180,E1 -8520.009,E2 -8520.009} C_VEL
LIN {X 0,Y 598.457,Z 282.495,A -85,B 0,C 180,E1 -8522.083,E2 -8522.083} C_VEL
LIN {X 0,Y 598.474,Z 282.494,A -85,B 0,C 180,E1 -8525.08,E2 -8525.08} C_VEL
LIN {X 0,Y 598.519,Z 282.488,A -85,B 0,C 180,E1 -8528.006,E2 -8528.006} C_VEL
LIN {X 0,Y 598.512,Z 282.489,A -85,B 0,C 180,E1 -8530.87,E2 -8530.87} C_VEL
LIN {X 0,Y 598.549,Z 282.483,A -85,B 0,C 180,E1 -8533.687,E2 -8533.687} C_VEL
LIN {X 0,Y 598.561,Z 282.483,A -85,B 0,C 180,E1 -8536.463,E2 -8536.463} C_VEL
LIN {X 0,Y 598.569,Z 282.48,A -85,B 0,C 180,E1 -8539.41,E2 -8539.41} C_VEL
LIN {X 0,Y 598.587,Z 282.481,A -85,B 0,C 180,E1 -8542.603,E2 -8542.603} C_VEL
LIN {X 0,Y 598.638,Z 282.501,A -85,B 0,C 180,E1 -8543.418,E2 -8543.418} C_VEL
LIN {X 0,Y 599.544,Z 289.354,A -85,B 0,C 180,E1 -8544.636,E2 -8544.636} C_VEL
LIN {X 0,Y 599.351,Z 298.165,A -85,B 0,C 180,E1 -8546.145,E2 -8546.145} C_VEL
LIN {X 0,Y 602.225,Z 312.367,A -85,B 0,C 180,E1 -8546.393,E2 -8546.393} C_VEL
LIN {X 0,Y 601.341,Z 433.246,A -85,B 0,C 180,E1 -8547.85,E2 -8547.85} C_VEL
LIN {X 0,Y 601.149,Z 447.755,A -85,B 0,C 180,E1 -8548.162,E2 -8548.162} C_VEL
LIN {X 0,Y 600.87,Z 461.046,A -85,B 0,C 180,E1 -8548.579,E2 -8548.579} C_VEL
LIN {X 0,Y 600.523,Z 473.183,A -85,B 0,C 180,E1 -8549.079,E2 -8549.079} C_VEL
LIN {X 0,Y 600.167,Z 485.898,A -85,B 0,C 180,E1 -8549.748,E2 -8549.748} C_VEL
LIN {X 0,Y 599.64,Z 497.516,A -85,B 0,C 180,E1 -8550.5,E2 -8550.5} C_VEL
LIN {X 0,Y 599.292,Z 508.113,A -85,B 0,C 180,E1 -8551.338,E2 -8551.338} C_VEL
LIN {X 0,Y 598.799,Z 518.653,A -85,B 0,C 180,E1 -8552.345,E2 -8552.345} C_VEL
LIN {X 0,Y 598.496,Z 527.348,A -85,B 0,C 180,E1 -8553.353,E2 -8553.353} C_VEL
LIN {X 0,Y 598.142,Z 534.617,A -85,B 0,C 180,E1 -8554.364,E2 -8554.364} C_VEL
LIN {X 0,Y 598.041,Z 540.836,A -85,B 0,C 180,E1 -8555.409,E2 -8555.409} C_VEL
LIN {X 0,Y 597.8,Z 547.109,A -85,B 0,C 180,E1 -8556.727,E2 -8556.727} C_VEL
LIN {X 0,Y 597.596,Z 551.95,A -85,B 0,C 180,E1 -8558.084,E2 -8558.084} C_VEL
LIN {X 0,Y 597.532,Z 555.306,A -85,B 0,C 180,E1 -8559.444,E2 -8559.444} C_VEL
LIN {X 0,Y 597.489,Z 557.269,A -85,B 0,C 180,E1 -8560.809,E2 -8560.809} C_VEL
LIN {X 0,Y 597.46,Z 557.867,A -85,B 0,C 180,E1 -8562.181,E2 -8562.181} C_VEL
LIN {X 0,Y 597.528,Z 557.104,A -85,B 0,C 180,E1 -8563.557,E2 -8563.557} C_VEL
LIN {X 0,Y 597.548,Z 554.957,A -85,B 0,C 180,E1 -8564.943,E2 -8564.943} C_VEL
LIN {X 0,Y 597.702,Z 551.345,A -85,B 0,C 180,E1 -8566.333,E2 -8566.333} C_VEL
LIN {X 0,Y 597.888,Z 546.142,A -85,B 0,C 180,E1 -8567.732,E2 -8567.732} C_VEL
LIN {X 0,Y 598.121,Z 541.031,A -85,B 0,C 180,E1 -8568.785,E2 -8568.785} C_VEL
LIN {X 0,Y 598.4,Z 533.633,A -85,B 0,C 180,E1 -8570.02,E2 -8570.02} C_VEL
LIN {X 0,Y 598.741,Z 525.791,A -85,B 0,C 180,E1 -8571.081,E2 -8571.081} C_VEL
LIN {X 0,Y 599.239,Z 516.386,A -85,B 0,C 180,E1 -8572.133,E2 -8572.133} C_VEL
LIN {X 0,Y 599.647,Z 505.597,A -85,B 0,C 180,E1 -8573.125,E2 -8573.125} C_VEL
LIN {X 0,Y 600.202,Z 493.678,A -85,B 0,C 180,E1 -8574.014,E2 -8574.014} C_VEL
LIN {X 0,Y 600.63,Z 481.307,A -85,B 0,C 180,E1 -8574.764,E2 -8574.764} C_VEL
LIN {X 0,Y 601.09,Z 468.066,A -85,B 0,C 180,E1 -8575.4,E2 -8575.4} C_VEL
LIN {X 0,Y 601.479,Z 454.696,A -85,B 0,C 180,E1 -8575.891,E2 -8575.891} C_VEL
LIN {X 0,Y 601.708,Z 441.218,A -85,B 0,C 180,E1 -8576.252,E2 -8576.252} C_VEL
LIN {X 0,Y 601.811,Z 427.48,A -85,B 0,C 180,E1 -8576.49,E2 -8576.49} C_VEL
LIN {X 0,Y 602.63,Z 312.009,A -85,B 0,C 180,E1 -8577.886,E2 -8577.886} C_VEL
LIN {X 0,Y 599.746,Z 298.528,A -85,B 0,C 180,E1 -8578.153,E2 -8578.153} C_VEL
LIN {X 0,Y 599.858,Z 290.536,A -85,B 0,C 180,E1 -8579.554,E2 -8579.554} C_VEL
LIN {X 0,Y 598.465,Z 282.498,A -85,B 0,C 180,E1 -8581.071,E2 -8581.071} C_VEL
LIN {X 0,Y 598.444,Z 282.499,A -85,B 0,C 180,E1 -8583.797,E2 -8583.797} C_VEL
LIN {X 0,Y 598.476,Z 282.493,A -85,B 0,C 180,E1 -8586.645,E2 -8586.645} C_VEL
LIN {X 0,Y 598.442,Z 282.494,A -85,B 0,C 180,E1 -8589.422,E2 -8589.422} C_VEL
LIN {X 0,Y 598.431,Z 282.497,A -85,B 0,C 180,E1 -8591.846,E2 -8591.846} C_VEL
LIN {X 0,Y 598.443,Z 282.488,A -85,B 0,C 180,E1 -8594.606,E2 -8594.606} C_VEL
LIN {X 0,Y 598.441,Z 282.498,A -85,B 0,C 180,E1 -8597.505,E2 -8597.505} C_VEL
LIN {X 0,Y 598.452,Z 282.499,A -85,B 0,C 180,E1 -8599.929,E2 -8599.929} C_VEL
LIN {X 0,Y 598.461,Z 282.489,A -85,B 0,C 180,E1 -8602.734,E2 -8602.734} C_VEL
LIN {X 0,Y 598.48,Z 282.479,A -85,B 0,C 180,E1 -8605.007,E2 -8605.007} C_VEL
LIN {X 0,Y 598.438,Z 282.498,A -85,B 0,C 180,E1 -8607.425,E2 -8607.425} C_VEL
LIN {X 0,Y 598.478,Z 282.494,A -85,B 0,C 180,E1 -8610.001,E2 -8610.001} C_VEL
LIN {X 0,Y 598.451,Z 282.491,A -85,B 0,C 180,E1 -8612.084,E2 -8612.084} C_VEL
LIN {X 0,Y 598.451,Z 282.495,A -85,B 0,C 180,E1 -8615.08,E2 -8615.08} C_VEL
LIN {X 0,Y 598.489,Z 282.493,A -85,B 0,C 180,E1 -8617.599,E2 -8617.599} C_VEL
LIN {X 0,Y 598.474,Z 282.487,A -85,B 0,C 180,E1 -8620.159,E2 -8620.159} C_VEL
LIN {X 0,Y 598.466,Z 282.492,A -85,B 0,C 180,E1 -8622.986,E2 -8622.986} C_VEL
LIN {X 0,Y 598.523,Z 282.482,A -85,B 0,C 180,E1 -8625.773,E2 -8625.773} C_VEL
LIN {X 0,Y 598.498,Z 282.487,A -85,B 0,C 180,E1 -8628.524,E2 -8628.524} C_VEL
LIN {X 0,Y 598.502,Z 282.483,A -85,B 0,C 180,E1 -8630.57,E2 -8630.57} C_VEL
LIN {X 0,Y 598.593,Z 282.484,A -85,B 0,C 180,E1 -8633.28,E2 -8633.28} C_VEL
LIN {X 0,Y 598.632,Z 282.463,A -85,B 0,C 180,E1 -8635.974,E2 -8635.974} C_VEL
LIN {X 0,Y 598.745,Z 282.461,A -85,B 0,C 180,E1 -8639.33,E2 -8639.33} C_VEL
LIN {X 0,Y 598.753,Z 282.452,A -85,B 0,C 180,E1 -8641.341,E2 -8641.341} C_VEL
LIN {X 0,Y 598.635,Z 282.473,A -85,B 0,C 180,E1 -8644.698,E2 -8644.698} C_VEL
LIN {X 0,Y 598.593,Z 282.478,A -85,B 0,C 180,E1 -8646.72,E2 -8646.72} C_VEL
LIN {X 0,Y 598.514,Z 282.486,A -85,B 0,C 180,E1 -8649.43,E2 -8649.43} C_VEL
LIN {X 0,Y 598.518,Z 282.48,A -85,B 0,C 180,E1 -8651.476,E2 -8651.476} C_VEL
LIN {X 0,Y 598.524,Z 282.481,A -85,B 0,C 180,E1 -8654.227,E2 -8654.227} C_VEL
LIN {X 0,Y 598.518,Z 282.483,A -85,B 0,C 180,E1 -8657.012,E2 -8657.012} C_VEL
LIN {X 0,Y 598.483,Z 282.487,A -85,B 0,C 180,E1 -8659.841,E2 -8659.841} C_VEL
LIN {X 0,Y 598.489,Z 282.488,A -85,B 0,C 180,E1 -8662.402,E2 -8662.402} C_VEL
LIN {X 0,Y 598.452,Z 282.495,A -85,B 0,C 180,E1 -8664.92,E2 -8664.92} C_VEL
LIN {X 0,Y 598.463,Z 282.491,A -85,B 0,C 180,E1 -8667.915,E2 -8667.915} C_VEL
LIN {X 0,Y 598.478,Z 282.493,A -85,B 0,C 180,E1 -8670.216,E2 -8670.216} C_VEL
LIN {X 0,Y 598.46,Z 282.498,A -85,B 0,C 180,E1 -8672.579,E2 -8672.579} C_VEL
LIN {X 0,Y 598.503,Z 282.474,A -85,B 0,C 180,E1 -8674.997,E2 -8674.997} C_VEL
LIN {X 0,Y 598.503,Z 282.482,A -85,B 0,C 180,E1 -8677.486,E2 -8677.486} C_VEL
LIN {X 0,Y 598.484,Z 282.495,A -85,B 0,C 180,E1 -8680.474,E2 -8680.474} C_VEL
LIN {X 0,Y 598.458,Z 282.493,A -85,B 0,C 180,E1 -8682.753,E2 -8682.753} C_VEL
LIN {X 0,Y 598.459,Z 282.491,A -85,B 0,C 180,E1 -8685.557,E2 -8685.557} C_VEL
LIN {X 0,Y 598.494,Z 282.491,A -85,B 0,C 180,E1 -8688.506,E2 -8688.506} C_VEL
LIN {X 0,Y 598.48,Z 282.49,A -85,B 0,C 180,E1 -8690.805,E2 -8690.805} C_VEL
LIN {X 0,Y 598.532,Z 282.483,A -85,B 0,C 180,E1 -8693.359,E2 -8693.359} C_VEL
LIN {X 0,Y 598.467,Z 282.5,A -85,B 0,C 180,E1 -8695.823,E2 -8695.823} C_VEL
LIN {X 0,Y 598.48,Z 282.495,A -85,B 0,C 180,E1 -8698.69,E2 -8698.69} C_VEL
LIN {X 0,Y 598.51,Z 282.491,A -85,B 0,C 180,E1 -8701.371,E2 -8701.371} C_VEL
LIN {X 0,Y 598.455,Z 282.509,A -85,B 0,C 180,E1 -8703.639,E2 -8703.639} C_VEL
LIN {X 0,Y 601.507,Z 296.847,A -85,B 0,C 180,E1 -8705.644,E2 -8705.644} C_VEL
LIN {X 0,Y 601.553,Z 302.061,A -85,B 0,C 180,E1 -8706.317,E2 -8706.317} C_VEL
LIN {X 0,Y 600.585,Z 323.582,A -85,B 0,C 180,E1 -8709.012,E2 -8709.012} C_VEL
LIN {X 0,Y 599.77,Z 344.73,A -85,B 0,C 180,E1 -8711.622,E2 -8711.622} C_VEL
LIN {X 0,Y 599.196,Z 363.185,A -85,B 0,C 180,E1 -8713.872,E2 -8713.872} C_VEL
LIN {X 0,Y 602.306,Z 386.134,A -85,B 0,C 180,E1 -8714.25,E2 -8714.25} C_VEL
LIN {X 0,Y 601.497,Z 501.478,A -85,B 0,C 180,E1 -8715.655,E2 -8715.655} C_VEL
LIN {X 0,Y 601.1,Z 515.965,A -85,B 0,C 180,E1 -8715.966,E2 -8715.966} C_VEL
LIN {X 0,Y 600.637,Z 529.354,A -85,B 0,C 180,E1 -8716.386,E2 -8716.386} C_VEL
LIN {X 0,Y 600.156,Z 542.474,A -85,B 0,C 180,E1 -8716.933,E2 -8716.933} C_VEL
LIN {X 0,Y 599.607,Z 555.171,A -85,B 0,C 180,E1 -8717.607,E2 -8717.607} C_VEL
LIN {X 0,Y 599.1,Z 566.751,A -85,B 0,C 180,E1 -8718.367,E2 -8718.367} C_VEL
LIN {X 0,Y 598.725,Z 577.397,A -85,B 0,C 180,E1 -8719.213,E2 -8719.213} C_VEL
LIN {X 0,Y 598.262,Z 587.982,A -85,B 0,C 180,E1 -8720.228,E2 -8720.228} C_VEL
LIN {X 0,Y 597.979,Z 596.743,A -85,B 0,C 180,E1 -8721.243,E2 -8721.243} C_VEL
LIN {X 0,Y 597.7,Z 605.168,A -85,B 0,C 180,E1 -8722.426,E2 -8722.426} C_VEL
LIN {X 0,Y 597.583,Z 612.185,A -85,B 0,C 180,E1 -8723.608,E2 -8723.608} C_VEL
LIN {X 0,Y 597.479,Z 617.193,A -85,B 0,C 180,E1 -8724.62,E2 -8724.62} C_VEL
LIN {X 0,Y 597.463,Z 622.324,A -85,B 0,C 180,E1 -8725.968,E2 -8725.968} C_VEL
LIN {X 0,Y 597.421,Z 625.897,A -85,B 0,C 180,E1 -8727.314,E2 -8727.314} C_VEL
LIN {X 0,Y 597.443,Z 628.022,A -85,B 0,C 180,E1 -8728.658,E2 -8728.658} C_VEL
LIN {X 0,Y 597.473,Z 628.745,A -85,B 0,C 180,E1 -8730.002,E2 -8730.002} C_VEL
LIN {X 0,Y 597.443,Z 628.057,A -85,B 0,C 180,E1 -8731.345,E2 -8731.345} C_VEL
LIN {X 0,Y 597.424,Z 625.955,A -85,B 0,C 180,E1 -8732.69,E2 -8732.69} C_VEL
LIN {X 0,Y 597.464,Z 622.404,A -85,B 0,C 180,E1 -8734.035,E2 -8734.035} C_VEL
LIN {X 0,Y 597.484,Z 617.294,A -85,B 0,C 180,E1 -8735.383,E2 -8735.383} C_VEL
LIN {X 0,Y 597.584,Z 612.329,A -85,B 0,C 180,E1 -8736.395,E2 -8736.395} C_VEL
LIN {X 0,Y 597.696,Z 605.152,A -85,B 0,C 180,E1 -8737.577,E2 -8737.577} C_VEL
LIN {X 0,Y 597.976,Z 596.252,A -85,B 0,C 180,E1 -8738.76,E2 -8738.76} C_VEL
LIN {X 0,Y 598.338,Z 585.467,A -85,B 0,C 180,E1 -8739.945,E2 -8739.945} C_VEL
LIN {X 0,Y 598.69,Z 575.268,A -85,B 0,C 180,E1 -8740.876,E2 -8740.876} C_VEL
LIN {X 0,Y 599.052,Z 564.066,A -85,B 0,C 180,E1 -8741.723,E2 -8741.723} C_VEL
LIN {X 0,Y 599.582,Z 551.714,A -85,B 0,C 180,E1 -8742.483,E2 -8742.483} C_VEL
LIN {X 0,Y 600.044,Z 539.858,A -85,B 0,C 180,E1 -8743.073,E2 -8743.073} C_VEL
LIN {X 0,Y 600.45,Z 526.933,A -85,B 0,C 180,E1 -8743.579,E2 -8743.579} C_VEL
LIN {X 0,Y 600.838,Z 513.127,A -85,B 0,C 180,E1 -8743.979,E2 -8743.979} C_VEL
LIN {X 0,Y 601.146,Z 499.609,A -85,B 0,C 180,E1 -8744.241,E2 -8744.241} C_VEL
LIN {X 0,Y 601.921,Z 386.264,A -85,B 0,C 180,E1 -8745.601,E2 -8745.601} C_VEL
LIN {X 0,Y 599.077,Z 363.318,A -85,B 0,C 180,E1 -8745.971,E2 -8745.971} C_VEL
LIN {X 0,Y 599.85,Z 335.978,A -85,B 0,C 180,E1 -8749.263,E2 -8749.263} C_VEL
LIN {X 0,Y 600.549,Z 315.612,A -85,B 0,C 180,E1 -8751.736,E2 -8751.736} C_VEL
LIN {X 0,Y 601.242,Z 296.669,A -85,B 0,C 180,E1 -8754.065,E2 -8754.065} C_VEL
LIN {X 0,Y 598.485,Z 282.497,A -85,B 0,C 180,E1 -8755.957,E2 -8755.957} C_VEL
LIN {X 0,Y 598.482,Z 282.491,A -85,B 0,C 180,E1 -8758.677,E2 -8758.677} C_VEL
LIN {X 0,Y 598.463,Z 282.495,A -85,B 0,C 180,E1 -8761.307,E2 -8761.307} C_VEL
LIN {X 0,Y 598.457,Z 282.496,A -85,B 0,C 180,E1 -8764.182,E2 -8764.182} C_VEL
LIN {X 0,Y 598.472,Z 282.491,A -85,B 0,C 180,E1 -8766.649,E2 -8766.649} C_VEL
LIN {X 0,Y 598.459,Z 282.499,A -85,B 0,C 180,E1 -8769.423,E2 -8769.423} C_VEL
LIN {X 0,Y 598.447,Z 282.495,A -85,B 0,C 180,E1 -8771.849,E2 -8771.849} C_VEL
LIN {X 0,Y 598.461,Z 282.493,A -85,B 0,C 180,E1 -8774.609,E2 -8774.609} C_VEL
LIN {X 0,Y 598.431,Z 282.499,A -85,B 0,C 180,E1 -8777.511,E2 -8777.511} C_VEL
LIN {X 0,Y 598.453,Z 282.492,A -85,B 0,C 180,E1 -8779.929,E2 -8779.929} C_VEL
LIN {X 0,Y 598.451,Z 282.5,A -85,B 0,C 180,E1 -8782.741,E2 -8782.741} C_VEL
LIN {X 0,Y 598.508,Z 282.492,A -85,B 0,C 180,E1 -8785.008,E2 -8785.008} C_VEL
LIN {X 0,Y 598.467,Z 282.492,A -85,B 0,C 180,E1 -8787.426,E2 -8787.426} C_VEL
LIN {X 0,Y 598.467,Z 282.495,A -85,B 0,C 180,E1 -8790.01,E2 -8790.01} C_VEL
LIN {X 0,Y 598.457,Z 282.497,A -85,B 0,C 180,E1 -8792.085,E2 -8792.085} C_VEL
LIN {X 0,Y 598.476,Z 282.493,A -85,B 0,C 180,E1 -8795.081,E2 -8795.081} C_VEL
LIN {X 0,Y 598.521,Z 282.496,A -85,B 0,C 180,E1 -8798.007,E2 -8798.007} C_VEL
LIN {X 0,Y 598.504,Z 282.499,A -85,B 0,C 180,E1 -8800.16,E2 -8800.16} C_VEL
LIN {X 0,Y 598.494,Z 282.491,A -85,B 0,C 180,E1 -8802.987,E2 -8802.987} C_VEL
LIN {X 0,Y 598.524,Z 282.493,A -85,B 0,C 180,E1 -8805.773,E2 -8805.773} C_VEL
LIN {X 0,Y 598.579,Z 282.618,A -85,B 0,C 180,E1 -8808.397,E2 -8808.397} C_VEL
LIN {X 0,Y 600.728,Z 294.228,A -85,B 0,C 180,E1 -8809.927,E2 -8809.927} C_VEL
LIN {X 0,Y 600.437,Z 315.888,A -85,B 0,C 180,E1 -8812.627,E2 -8812.627} C_VEL
LIN {X 0,Y 599.769,Z 342.521,A -85,B 0,C 180,E1 -8815.94,E2 -8815.94} C_VEL
LIN {X 0,Y 602.458,Z 358.034,A -85,B 0,C 180,E1 -8816.25,E2 -8816.25} C_VEL
LIN {X 0,Y 601.123,Z 480.571,A -85,B 0,C 180,E1 -8817.913,E2 -8817.913} C_VEL
LIN {X 0,Y 600.843,Z 495.335,A -85,B 0,C 180,E1 -8818.246,E2 -8818.246} C_VEL
LIN {X 0,Y 600.44,Z 509.294,A -85,B 0,C 180,E1 -8818.705,E2 -8818.705} C_VEL
LIN {X 0,Y 600.044,Z 521.831,A -85,B 0,C 180,E1 -8819.248,E2 -8819.248} C_VEL
LIN {X 0,Y 599.574,Z 534.132,A -85,B 0,C 180,E1 -8819.916,E2 -8819.916} C_VEL
LIN {X 0,Y 599.241,Z 546.513,A -85,B 0,C 180,E1 -8820.753,E2 -8820.753} C_VEL
LIN {X 0,Y 598.764,Z 557.724,A -85,B 0,C 180,E1 -8821.676,E2 -8821.676} C_VEL
LIN {X 0,Y 598.318,Z 567.808,A -85,B 0,C 180,E1 -8822.684,E2 -8822.684} C_VEL
LIN {X 0,Y 597.999,Z 576.149,A -85,B 0,C 180,E1 -8823.694,E2 -8823.694} C_VEL
LIN {X 0,Y 597.793,Z 584.017,A -85,B 0,C 180,E1 -8824.857,E2 -8824.857} C_VEL
LIN {X 0,Y 597.669,Z 590.532,A -85,B 0,C 180,E1 -8826.055,E2 -8826.055} C_VEL
LIN {X 0,Y 597.5,Z 596.231,A -85,B 0,C 180,E1 -8827.409,E2 -8827.409} C_VEL
LIN {X 0,Y 597.409,Z 600.36,A -85,B 0,C 180,E1 -8828.767,E2 -8828.767} C_VEL
LIN {X 0,Y 597.39,Z 603.008,A -85,B 0,C 180,E1 -8830.13,E2 -8830.13} C_VEL
LIN {X 0,Y 597.294,Z 604.208,A -85,B 0,C 180,E1 -8831.499,E2 -8831.499} C_VEL
LIN {X 0,Y 597.357,Z 603.993,A -85,B 0,C 180,E1 -8832.873,E2 -8832.873} C_VEL
LIN {X 0,Y 597.352,Z 602.35,A -85,B 0,C 180,E1 -8834.255,E2 -8834.255} C_VEL
LIN {X 0,Y 597.43,Z 599.227,A -85,B 0,C 180,E1 -8835.644,E2 -8835.644} C_VEL
LIN {X 0,Y 597.476,Z 595.811,A -85,B 0,C 180,E1 -8836.692,E2 -8836.692} C_VEL
LIN {X 0,Y 597.625,Z 590.049,A -85,B 0,C 180,E1 -8838.032,E2 -8838.032} C_VEL
LIN {X 0,Y 597.842,Z 582.782,A -85,B 0,C 180,E1 -8839.328,E2 -8839.328} C_VEL
LIN {X 0,Y 598.076,Z 574.867,A -85,B 0,C 180,E1 -8840.456,E2 -8840.456} C_VEL
LIN {X 0,Y 598.364,Z 566.35,A -85,B 0,C 180,E1 -8841.458,E2 -8841.458} C_VEL
LIN {X 0,Y 598.761,Z 556.102,A -85,B 0,C 180,E1 -8842.456,E2 -8842.456} C_VEL
LIN {X 0,Y 599.115,Z 545.255,A -85,B 0,C 180,E1 -8843.331,E2 -8843.331} C_VEL
LIN {X 0,Y 599.605,Z 533.125,A -85,B 0,C 180,E1 -8844.133,E2 -8844.133} C_VEL
LIN {X 0,Y 599.915,Z 521.121,A -85,B 0,C 180,E1 -8844.78,E2 -8844.78} C_VEL
LIN {X 0,Y 600.297,Z 507.826,A -85,B 0,C 180,E1 -8845.346,E2 -8845.346} C_VEL
LIN {X 0,Y 600.665,Z 493.577,A -85,B 0,C 180,E1 -8845.796,E2 -8845.796} C_VEL
LIN {X 0,Y 600.94,Z 478.8,A -85,B 0,C 180,E1 -8846.115,E2 -8846.115} C_VEL
LIN {X 0,Y 602.044,Z 357.972,A -85,B 0,C 180,E1 -8847.694,E2 -8847.694} C_VEL
LIN {X 0,Y 599.485,Z 341.75,A -85,B 0,C 180,E1 -8847.993,E2 -8847.993} C_VEL
LIN {X 0,Y 599.974,Z 320.348,A -85,B 0,C 180,E1 -8850.717,E2 -8850.717} C_VEL
LIN {X 0,Y 600.555,Z 297.383,A -85,B 0,C 180,E1 -8853.642,E2 -8853.642} C_VEL
LIN {X 0,Y 600.392,Z 292.632,A -85,B 0,C 180,E1 -8854.257,E2 -8854.257} C_VEL
LIN {X 0,Y 598.539,Z 282.488,A -85,B 0,C 180,E1 -8855.621,E2 -8855.621} C_VEL
LIN {X 0,Y 598.465,Z 282.499,A -85,B 0,C 180,E1 -8858.355,E2 -8858.355} C_VEL
LIN {X 0,Y 598.472,Z 282.491,A -85,B 0,C 180,E1 -8860.951,E2 -8860.951} C_VEL
LIN {X 0,Y 598.461,Z 282.495,A -85,B 0,C 180,E1 -8863.673,E2 -8863.673} C_VEL
LIN {X 0,Y 598.458,Z 282.495,A -85,B 0,C 180,E1 -8866.524,E2 -8866.524} C_VEL
LIN {X 0,Y 598.475,Z 282.494,A -85,B 0,C 180,E1 -8869.53,E2 -8869.53} C_VEL
LIN {X 0,Y 598.454,Z 282.499,A -85,B 0,C 180,E1 -8870.012,E2 -8870.012} C_VEL
LIN {X 0,Y 597.779,Z 282.579,A -85,B 0,C 180,E1 -8870.573,E2 -8870.573} C_VEL
LIN {X 0,Y 594.922,Z 282.937,A -85,B 0,C 180,E1 -8871.485,E2 -8871.485} C_VEL
LIN {X 0,Y 592.512,Z 283.238,A -85,B 0,C 180,E1 -8872.219,E2 -8872.219} C_VEL
LIN {X 0,Y 591.475,Z 283.366,A -85,B 0,C 180,E1 -8872.785,E2 -8872.785} C_VEL
LIN {X 0,Y 591.389,Z 283.376,A -85,B 0,C 180,E1 -8872.976,E2 -8872.976} C_VEL
LIN {X 0,Y 591.401,Z 283.376,A -85,B 0,C 180,E1 -8875.353,E2 -8875.353} C_VEL
LIN {X 0,Y 591.415,Z 283.374,A -85,B 0,C 180,E1 -8877.793,E2 -8877.793} C_VEL
LIN {X 0,Y 591.414,Z 283.372,A -85,B 0,C 180,E1 -8880.169,E2 -8880.169} C_VEL
LIN {X 0,Y 591.431,Z 283.374,A -85,B 0,C 180,E1 -8882.653,E2 -8882.653} C_VEL
LIN {X 0,Y 591.443,Z 283.368,A -85,B 0,C 180,E1 -8885.771,E2 -8885.771} C_VEL
LIN {X 0,Y 591.478,Z 283.368,A -85,B 0,C 180,E1 -8888.461,E2 -8888.461} C_VEL
LIN {X 0,Y 591.479,Z 283.364,A -85,B 0,C 180,E1 -8891.351,E2 -8891.351} C_VEL
LIN {X 0,Y 591.492,Z 283.368,A -85,B 0,C 180,E1 -8894.193,E2 -8894.193} C_VEL
LIN {X 0,Y 591.513,Z 283.363,A -85,B 0,C 180,E1 -8896.299,E2 -8896.299} C_VEL
LIN {X 0,Y 591.541,Z 283.355,A -85,B 0,C 180,E1 -8899.359,E2 -8899.359} C_VEL
LIN {X 0,Y 591.55,Z 283.358,A -85,B 0,C 180,E1 -8902.514,E2 -8902.514} C_VEL
LIN {X 0,Y 591.59,Z 283.472,A -85,B 0,C 180,E1 -8903.327,E2 -8903.327} C_VEL
LIN {X 0,Y 592.549,Z 290.416,A -85,B 0,C 180,E1 -8904.572,E2 -8904.572} C_VEL
LIN {X 0,Y 592.326,Z 298.543,A -85,B 0,C 180,E1 -8905.972,E2 -8905.972} C_VEL
LIN {X 0,Y 595.273,Z 312.594,A -85,B 0,C 180,E1 -8906.224,E2 -8906.224} C_VEL
LIN {X 0,Y 594.425,Z 433.434,A -85,B 0,C 180,E1 -8907.698,E2 -8907.698} C_VEL
LIN {X 0,Y 594.226,Z 448.036,A -85,B 0,C 180,E1 -8908.014,E2 -8908.014} C_VEL
LIN {X 0,Y 593.938,Z 461.364,A -85,B 0,C 180,E1 -8908.436,E2 -8908.436} C_VEL
LIN {X 0,Y 593.553,Z 474.393,A -85,B 0,C 180,E1 -8908.984,E2 -8908.984} C_VEL
LIN {X 0,Y 593.197,Z 486.955,A -85,B 0,C 180,E1 -8909.66,E2 -8909.66} C_VEL
LIN {X 0,Y 592.638,Z 498.468,A -85,B 0,C 180,E1 -8910.422,E2 -8910.422} C_VEL
LIN {X 0,Y 592.248,Z 509.938,A -85,B 0,C 180,E1 -8911.354,E2 -8911.354} C_VEL
LIN {X 0,Y 591.732,Z 520.248,A -85,B 0,C 180,E1 -8912.373,E2 -8912.373} C_VEL
LIN {X 0,Y 591.428,Z 528.745,A -85,B 0,C 180,E1 -8913.393,E2 -8913.393} C_VEL
LIN {X 0,Y 591.025,Z 536.932,A -85,B 0,C 180,E1 -8914.587,E2 -8914.587} C_VEL
LIN {X 0,Y 590.884,Z 543.498,A -85,B 0,C 180,E1 -8915.781,E2 -8915.781} C_VEL
LIN {X 0,Y 590.667,Z 549.353,A -85,B 0,C 180,E1 -8917.151,E2 -8917.151} C_VEL
LIN {X 0,Y 590.506,Z 552.754,A -85,B 0,C 180,E1 -8918.182,E2 -8918.182} C_VEL
LIN {X 0,Y 590.456,Z 555.954,A -85,B 0,C 180,E1 -8919.558,E2 -8919.558} C_VEL
LIN {X 0,Y 590.39,Z 557.777,A -85,B 0,C 180,E1 -8920.941,E2 -8920.941} C_VEL
LIN {X 0,Y 590.401,Z 558.251,A -85,B 0,C 180,E1 -8922.329,E2 -8922.329} C_VEL
LIN {X 0,Y 590.446,Z 557.37,A -85,B 0,C 180,E1 -8923.723,E2 -8923.723} C_VEL
LIN {X 0,Y 590.484,Z 555.1,A -85,B 0,C 180,E1 -8925.126,E2 -8925.126} C_VEL
LIN {X 0,Y 590.658,Z 551.36,A -85,B 0,C 180,E1 -8926.533,E2 -8926.533} C_VEL
LIN {X 0,Y 590.803,Z 547.473,A -85,B 0,C 180,E1 -8927.595,E2 -8927.595} C_VEL
LIN {X 0,Y 591.04,Z 542.614,A -85,B 0,C 180,E1 -8928.66,E2 -8928.66} C_VEL
LIN {X 0,Y 591.353,Z 535.496,A -85,B 0,C 180,E1 -8929.907,E2 -8929.907} C_VEL
LIN {X 0,Y 591.656,Z 527.968,A -85,B 0,C 180,E1 -8930.983,E2 -8930.983} C_VEL
LIN {X 0,Y 592.168,Z 518.829,A -85,B 0,C 180,E1 -8932.056,E2 -8932.056} C_VEL
LIN {X 0,Y 592.632,Z 508.64,A -85,B 0,C 180,E1 -8933.046,E2 -8933.046} C_VEL
LIN {X 0,Y 593.198,Z 497.377,A -85,B 0,C 180,E1 -8933.945,E2 -8933.945} C_VEL
LIN {X 0,Y 593.681,Z 484.826,A -85,B 0,C 180,E1 -8934.763,E2 -8934.763} C_VEL
LIN {X 0,Y 594.166,Z 471.704,A -85,B 0,C 180,E1 -8935.437,E2 -8935.437} C_VEL
LIN {X 0,Y 594.53,Z 458.147,A -85,B 0,C 180,E1 -8935.975,E2 -8935.975} C_VEL
LIN {X 0,Y 594.805,Z 443.845,A -85,B 0,C 180,E1 -8936.388,E2 -8936.388} C_VEL
LIN {X 0,Y 595,Z 428.892,A -85,B 0,C 180,E1 -8936.665,E2 -8936.665} C_VEL
LIN {X 0,Y 595.882,Z 312.985,A -85,B 0,C 180,E1 -8938.085,E2 -8938.085} C_VEL
LIN {X 0,Y 592.837,Z 298.892,A -85,B 0,C 180,E1 -8938.376,E2 -8938.376} C_VEL
LIN {X 0,Y 592.886,Z 291.206,A -85,B 0,C 180,E1 -8939.746,E2 -8939.746} C_VEL
LIN {X 0,Y 591.418,Z 283.376,A -85,B 0,C 180,E1 -8941.255,E2 -8941.255} C_VEL
LIN {X 0,Y 591.394,Z 283.38,A -85,B 0,C 180,E1 -8943.996,E2 -8943.996} C_VEL
LIN {X 0,Y 591.445,Z 283.374,A -85,B 0,C 180,E1 -8946.359,E2 -8946.359} C_VEL
LIN {X 0,Y 591.391,Z 283.372,A -85,B 0,C 180,E1 -8948.88,E2 -8948.88} C_VEL
LIN {X 0,Y 591.396,Z 283.373,A -85,B 0,C 180,E1 -8951.741,E2 -8951.741} C_VEL
LIN {X 0,Y 591.402,Z 283.364,A -85,B 0,C 180,E1 -8954.714,E2 -8954.714} C_VEL
LIN {X 0,Y 591.411,Z 283.374,A -85,B 0,C 180,E1 -8957.539,E2 -8957.539} C_VEL
LIN {X 0,Y 591.398,Z 283.374,A -85,B 0,C 180,E1 -8960.337,E2 -8960.337} C_VEL
LIN {X 0,Y 591.416,Z 283.366,A -85,B 0,C 180,E1 -8962.842,E2 -8962.842} C_VEL
LIN {X 0,Y 591.403,Z 283.363,A -85,B 0,C 180,E1 -8965.354,E2 -8965.354} C_VEL
LIN {X 0,Y 591.426,Z 283.365,A -85,B 0,C 180,E1 -8968.594,E2 -8968.594} C_VEL
LIN {X 0,Y 591.465,Z 283.365,A -85,B 0,C 180,E1 -8971.2,E2 -8971.2} C_VEL
LIN {X 0,Y 591.384,Z 283.375,A -85,B 0,C 180,E1 -8974.173,E2 -8974.173} C_VEL
LIN {X 0,Y 591.424,Z 283.364,A -85,B 0,C 180,E1 -8976.255,E2 -8976.255} C_VEL
LIN {X 0,Y 591.448,Z 283.365,A -85,B 0,C 180,E1 -8978.461,E2 -8978.461} C_VEL
LIN {X 0,Y 591.429,Z 283.369,A -85,B 0,C 180,E1 -8981.351,E2 -8981.351} C_VEL
LIN {X 0,Y 591.461,Z 283.362,A -85,B 0,C 180,E1 -8984.194,E2 -8984.194} C_VEL
LIN {X 0,Y 591.471,Z 283.36,A -85,B 0,C 180,E1 -8986.997,E2 -8986.997} C_VEL
LIN {X 0,Y 591.498,Z 283.357,A -85,B 0,C 180,E1 -8989.768,E2 -8989.768} C_VEL
LIN {X 0,Y 591.528,Z 283.353,A -85,B 0,C 180,E1 -8992.516,E2 -8992.516} C_VEL
LIN {X 0,Y 591.592,Z 283.349,A -85,B 0,C 180,E1 -8995.246,E2 -8995.246} C_VEL
LIN {X 0,Y 591.716,Z 283.337,A -85,B 0,C 180,E1 -8999.322,E2 -8999.322} C_VEL
LIN {X 0,Y 591.699,Z 283.331,A -85,B 0,C 180,E1 -9001.357,E2 -9001.357} C_VEL
LIN {X 0,Y 591.605,Z 283.35,A -85,B 0,C 180,E1 -9004.754,E2 -9004.754} C_VEL
LIN {X 0,Y 591.528,Z 283.351,A -85,B 0,C 180,E1 -9007.484,E2 -9007.484} C_VEL
LIN {X 0,Y 591.576,Z 283.353,A -85,B 0,C 180,E1 -9010.673,E2 -9010.673} C_VEL
LIN {X 0,Y 591.498,Z 283.355,A -85,B 0,C 180,E1 -9013.835,E2 -9013.835} C_VEL
LIN {X 0,Y 591.485,Z 283.363,A -85,B 0,C 180,E1 -9016.512,E2 -9016.512} C_VEL
LIN {X 0,Y 591.433,Z 283.367,A -85,B 0,C 180,E1 -9019.366,E2 -9019.366} C_VEL
LIN {X 0,Y 591.449,Z 283.36,A -85,B 0,C 180,E1 -9021.539,E2 -9021.539} C_VEL
LIN {X 0,Y 591.414,Z 283.375,A -85,B 0,C 180,E1 -9024.489,E2 -9024.489} C_VEL
LIN {X 0,Y 591.411,Z 283.368,A -85,B 0,C 180,E1 -9027.51,E2 -9027.51} C_VEL
LIN {X 0,Y 591.428,Z 283.367,A -85,B 0,C 180,E1 -9029.829,E2 -9029.829} C_VEL
LIN {X 0,Y 591.43,Z 283.372,A -85,B 0,C 180,E1 -9032.205,E2 -9032.205} C_VEL
LIN {X 0,Y 591.475,Z 283.347,A -85,B 0,C 180,E1 -9035.207,E2 -9035.207} C_VEL
LIN {X 0,Y 591.455,Z 283.364,A -85,B 0,C 180,E1 -9038.012,E2 -9038.012} C_VEL
LIN {X 0,Y 591.435,Z 283.37,A -85,B 0,C 180,E1 -9040.719,E2 -9040.719} C_VEL
LIN {X 0,Y 591.403,Z 283.37,A -85,B 0,C 180,E1 -9043.388,E2 -9043.388} C_VEL
LIN {X 0,Y 591.431,Z 283.376,A -85,B 0,C 180,E1 -9046.256,E2 -9046.256} C_VEL
LIN {X 0,Y 591.446,Z 283.37,A -85,B 0,C 180,E1 -9048.458,E2 -9048.458} C_VEL
LIN {X 0,Y 591.423,Z 283.369,A -85,B 0,C 180,E1 -9051.413,E2 -9051.413} C_VEL
LIN {X 0,Y 591.475,Z 283.364,A -85,B 0,C 180,E1 -9053.695,E2 -9053.695} C_VEL
LIN {X 0,Y 591.433,Z 283.373,A -85,B 0,C 180,E1 -9056.18,E2 -9056.18} C_VEL
LIN {X 0,Y 591.44,Z 283.373,A -85,B 0,C 180,E1 -9058.597,E2 -9058.597} C_VEL
LIN {X 0,Y 591.478,Z 283.366,A -85,B 0,C 180,E1 -9061.203,E2 -9061.203} C_VEL
LIN {X 0,Y 591.425,Z 283.482,A -85,B 0,C 180,E1 -9063.446,E2 -9063.446} C_VEL
LIN {X 0,Y 594.522,Z 297.919,A -85,B 0,C 180,E1 -9065.497,E2 -9065.497} C_VEL
LIN {X 0,Y 594.723,Z 301.93,A -85,B 0,C 180,E1 -9066.028,E2 -9066.028} C_VEL
LIN {X 0,Y 593.67,Z 324.248,A -85,B 0,C 180,E1 -9068.864,E2 -9068.864} C_VEL
LIN {X 0,Y 592.787,Z 345.946,A -85,B 0,C 180,E1 -9071.576,E2 -9071.576} C_VEL
LIN {X 0,Y 592.214,Z 362.755,A -85,B 0,C 180,E1 -9073.655,E2 -9073.655} C_VEL
LIN {X 0,Y 595.552,Z 387.438,A -85,B 0,C 180,E1 -9074.067,E2 -9074.067} C_VEL
LIN {X 0,Y 594.661,Z 501.619,A -85,B 0,C 180,E1 -9075.478,E2 -9075.478} C_VEL
LIN {X 0,Y 594.218,Z 516.229,A -85,B 0,C 180,E1 -9075.801,E2 -9075.801} C_VEL
LIN {X 0,Y 593.711,Z 530.557,A -85,B 0,C 180,E1 -9076.267,E2 -9076.267} C_VEL
LIN {X 0,Y 593.17,Z 544.196,A -85,B 0,C 180,E1 -9076.863,E2 -9076.863} C_VEL
LIN {X 0,Y 592.581,Z 556.473,A -85,B 0,C 180,E1 -9077.544,E2 -9077.544} C_VEL
LIN {X 0,Y 592.033,Z 568.905,A -85,B 0,C 180,E1 -9078.399,E2 -9078.399} C_VEL
LIN {X 0,Y 591.626,Z 579.77,A -85,B 0,C 180,E1 -9079.316,E2 -9079.316} C_VEL
LIN {X 0,Y 591.22,Z 589.31,A -85,B 0,C 180,E1 -9080.282,E2 -9080.282} C_VEL
LIN {X 0,Y 590.859,Z 597.779,A -85,B 0,C 180,E1 -9081.308,E2 -9081.308} C_VEL
LIN {X 0,Y 590.602,Z 605.903,A -85,B 0,C 180,E1 -9082.506,E2 -9082.506} C_VEL
LIN {X 0,Y 590.44,Z 613.746,A -85,B 0,C 180,E1 -9083.873,E2 -9083.873} C_VEL
LIN {X 0,Y 590.389,Z 618.407,A -85,B 0,C 180,E1 -9084.897,E2 -9084.897} C_VEL
LIN {X 0,Y 590.365,Z 622.118,A -85,B 0,C 180,E1 -9085.92,E2 -9085.92} C_VEL
LIN {X 0,Y 590.338,Z 625.715,A -85,B 0,C 180,E1 -9087.281,E2 -9087.281} C_VEL
LIN {X 0,Y 590.343,Z 627.858,A -85,B 0,C 180,E1 -9088.642,E2 -9088.642} C_VEL
LIN {X 0,Y 590.375,Z 628.596,A -85,B 0,C 180,E1 -9090.002,E2 -9090.002} C_VEL
LIN {X 0,Y 590.343,Z 627.921,A -85,B 0,C 180,E1 -9091.361,E2 -9091.361} C_VEL
LIN {X 0,Y 590.34,Z 625.824,A -85,B 0,C 180,E1 -9092.722,E2 -9092.722} C_VEL
LIN {X 0,Y 590.367,Z 622.273,A -85,B 0,C 180,E1 -9094.084,E2 -9094.084} C_VEL
LIN {X 0,Y 590.404,Z 617.168,A -85,B 0,C 180,E1 -9095.448,E2 -9095.448} C_VEL
LIN {X 0,Y 590.495,Z 612.208,A -85,B 0,C 180,E1 -9096.472,E2 -9096.472} C_VEL
LIN {X 0,Y 590.641,Z 605.039,A -85,B 0,C 180,E1 -9097.668,E2 -9097.668} C_VEL
LIN {X 0,Y 590.923,Z 596.135,A -85,B 0,C 180,E1 -9098.866,E2 -9098.866} C_VEL
LIN {X 0,Y 591.221,Z 586.768,A -85,B 0,C 180,E1 -9099.893,E2 -9099.893} C_VEL
LIN {X 0,Y 591.718,Z 573.623,A -85,B 0,C 180,E1 -9101.092,E2 -9101.092} C_VEL
LIN {X 0,Y 592.138,Z 562.101,A -85,B 0,C 180,E1 -9101.949,E2 -9101.949} C_VEL
LIN {X 0,Y 592.68,Z 549.372,A -85,B 0,C 180,E1 -9102.717,E2 -9102.717} C_VEL
LIN {X 0,Y 593.175,Z 537.016,A -85,B 0,C 180,E1 -9103.314,E2 -9103.314} C_VEL
LIN {X 0,Y 593.646,Z 523.349,A -85,B 0,C 180,E1 -9103.825,E2 -9103.825} C_VEL
LIN {X 0,Y 594.008,Z 509.166,A -85,B 0,C 180,E1 -9104.208,E2 -9104.208} C_VEL
LIN {X 0,Y 594.303,Z 494.651,A -85,B 0,C 180,E1 -9104.456,E2 -9104.456} C_VEL
LIN {X 0,Y 595.048,Z 386.898,A -85,B 0,C 180,E1 -9105.753,E2 -9105.753} C_VEL
LIN {X 0,Y 592.091,Z 362.375,A -85,B 0,C 180,E1 -9106.209,E2 -9106.209} C_VEL
LIN {X 0,Y 592.972,Z 333.954,A -85,B 0,C 180,E1 -9109.675,E2 -9109.675} C_VEL
LIN {X 0,Y 593.902,Z 309.22,A -85,B 0,C 180,E1 -9112.723,E2 -9112.723} C_VEL
LIN {X 0,Y 594.247,Z 297.548,A -85,B 0,C 180,E1 -9114.181,E2 -9114.181} C_VEL
LIN {X 0,Y 591.425,Z 283.376,A -85,B 0,C 180,E1 -9116.085,E2 -9116.085} C_VEL
LIN {X 0,Y 591.432,Z 283.369,A -85,B 0,C 180,E1 -9119.051,E2 -9119.051} C_VEL
LIN {X 0,Y 591.42,Z 283.375,A -85,B 0,C 180,E1 -9121.49,E2 -9121.49} C_VEL
LIN {X 0,Y 591.411,Z 283.376,A -85,B 0,C 180,E1 -9123.998,E2 -9123.998} C_VEL
LIN {X 0,Y 591.442,Z 283.368,A -85,B 0,C 180,E1 -9126.358,E2 -9126.358} C_VEL
LIN {X 0,Y 591.411,Z 283.373,A -85,B 0,C 180,E1 -9128.883,E2 -9128.883} C_VEL
LIN {X 0,Y 591.415,Z 283.372,A -85,B 0,C 180,E1 -9131.743,E2 -9131.743} C_VEL
LIN {X 0,Y 591.421,Z 283.371,A -85,B 0,C 180,E1 -9134.716,E2 -9134.716} C_VEL
LIN {X 0,Y 591.403,Z 283.374,A -85,B 0,C 180,E1 -9137.538,E2 -9137.538} C_VEL
LIN {X 0,Y 591.41,Z 283.371,A -85,B 0,C 180,E1 -9140.341,E2 -9140.341} C_VEL
LIN {X 0,Y 591.41,Z 283.377,A -85,B 0,C 180,E1 -9142.841,E2 -9142.841} C_VEL
LIN {X 0,Y 591.429,Z 283.369,A -85,B 0,C 180,E1 -9145.356,E2 -9145.356} C_VEL
LIN {X 0,Y 591.439,Z 283.374,A -85,B 0,C 180,E1 -9148.508,E2 -9148.508} C_VEL
LIN {X 0,Y 591.447,Z 283.366,A -85,B 0,C 180,E1 -9151.21,E2 -9151.21} C_VEL
LIN {X 0,Y 591.414,Z 283.377,A -85,B 0,C 180,E1 -9154.174,E2 -9154.174} C_VEL
LIN {X 0,Y 591.437,Z 283.371,A -85,B 0,C 180,E1 -9156.994,E2 -9156.994} C_VEL
LIN {X 0,Y 591.495,Z 283.366,A -85,B 0,C 180,E1 -9159.313,E2 -9159.313} C_VEL
LIN {X 0,Y 591.446,Z 283.377,A -85,B 0,C 180,E1 -9162.066,E2 -9162.066} C_VEL
LIN {X 0,Y 591.458,Z 283.368,A -85,B 0,C 180,E1 -9164.898,E2 -9164.898} C_VEL
LIN {X 0,Y 591.486,Z 283.367,A -85,B 0,C 180,E1 -9166.997,E2 -9166.997} C_VEL
LIN {X 0,Y 591.519,Z 283.425,A -85,B 0,C 180,E1 -9168.192,E2 -9168.192} C_VEL
LIN {X 0,Y 593.839,Z 295.532,A -85,B 0,C 180,E1 -9169.809,E2 -9169.809} C_VEL
LIN {X 0,Y 593.563,Z 316.414,A -85,B 0,C 180,E1 -9172.423,E2 -9172.423} C_VEL
LIN {X 0,Y 592.89,Z 342.847,A -85,B 0,C 180,E1 -9175.723,E2 -9175.723} C_VEL
LIN {X 0,Y 595.743,Z 359.384,A -85,B 0,C 180,E1 -9176.06,E2 -9176.06} C_VEL
LIN {X 0,Y 594.284,Z 480.82,A -85,B 0,C 180,E1 -9177.741,E2 -9177.741} C_VEL
LIN {X 0,Y 593.967,Z 495.52,A -85,B 0,C 180,E1 -9178.078,E2 -9178.078} C_VEL
LIN {X 0,Y 593.544,Z 509.968,A -85,B 0,C 180,E1 -9178.563,E2 -9178.563} C_VEL
LIN {X 0,Y 593.148,Z 521.576,A -85,B 0,C 180,E1 -9179.07,E2 -9179.07} C_VEL
LIN {X 0,Y 592.666,Z 533.954,A -85,B 0,C 180,E1 -9179.746,E2 -9179.746} C_VEL
LIN {X 0,Y 592.288,Z 546.398,A -85,B 0,C 180,E1 -9180.593,E2 -9180.593} C_VEL
LIN {X 0,Y 591.78,Z 557.648,A -85,B 0,C 180,E1 -9181.526,E2 -9181.526} C_VEL
LIN {X 0,Y 591.293,Z 567.775,A -85,B 0,C 180,E1 -9182.546,E2 -9182.546} C_VEL
LIN {X 0,Y 591.005,Z 576.136,A -85,B 0,C 180,E1 -9183.567,E2 -9183.567} C_VEL
LIN {X 0,Y 590.758,Z 584.148,A -85,B 0,C 180,E1 -9184.761,E2 -9184.761} C_VEL
LIN {X 0,Y 590.638,Z 589.786,A -85,B 0,C 180,E1 -9185.785,E2 -9185.785} C_VEL
LIN {X 0,Y 590.481,Z 594.375,A -85,B 0,C 180,E1 -9186.813,E2 -9186.813} C_VEL
LIN {X 0,Y 590.315,Z 599.12,A -85,B 0,C 180,E1 -9188.186,E2 -9188.186} C_VEL
LIN {X 0,Y 590.324,Z 602.295,A -85,B 0,C 180,E1 -9189.562,E2 -9189.562} C_VEL
LIN {X 0,Y 590.213,Z 604.045,A -85,B 0,C 180,E1 -9190.946,E2 -9190.946} C_VEL
LIN {X 0,Y 590.222,Z 604.384,A -85,B 0,C 180,E1 -9192.334,E2 -9192.334} C_VEL
LIN {X 0,Y 590.276,Z 603.302,A -85,B 0,C 180,E1 -9193.729,E2 -9193.729} C_VEL
LIN {X 0,Y 590.271,Z 600.763,A -85,B 0,C 180,E1 -9195.133,E2 -9195.133} C_VEL
LIN {X 0,Y 590.368,Z 598.251,A -85,B 0,C 180,E1 -9196.046,E2 -9196.046} C_VEL
LIN {X 0,Y 590.424,Z 593.913,A -85,B 0,C 180,E1 -9197.253,E2 -9197.253} C_VEL
LIN {X 0,Y 590.58,Z 588.537,A -85,B 0,C 180,E1 -9198.407,E2 -9198.407} C_VEL
LIN {X 0,Y 590.796,Z 581.78,A -85,B 0,C 180,E1 -9199.568,E2 -9199.568} C_VEL
LIN {X 0,Y 591.044,Z 574.695,A -85,B 0,C 180,E1 -9200.571,E2 -9200.571} C_VEL
LIN {X 0,Y 591.371,Z 564.798,A -85,B 0,C 180,E1 -9201.724,E2 -9201.724} C_VEL
LIN {X 0,Y 591.799,Z 554.323,A -85,B 0,C 180,E1 -9202.724,E2 -9202.724} C_VEL
LIN {X 0,Y 592.216,Z 542.927,A -85,B 0,C 180,E1 -9203.619,E2 -9203.619} C_VEL
LIN {X 0,Y 592.667,Z 530.091,A -85,B 0,C 180,E1 -9204.434,E2 -9204.434} C_VEL
LIN {X 0,Y 593.03,Z 517.65,A -85,B 0,C 180,E1 -9205.07,E2 -9205.07} C_VEL
LIN {X 0,Y 593.474,Z 504.071,A -85,B 0,C 180,E1 -9205.611,E2 -9205.611} C_VEL
LIN {X 0,Y 593.826,Z 489.83,A -85,B 0,C 180,E1 -9206.031,E2 -9206.031} C_VEL
LIN {X 0,Y 594.048,Z 475.683,A -85,B 0,C 180,E1 -9206.308,E2 -9206.308} C_VEL
LIN {X 0,Y 595.17,Z 358.745,A -85,B 0,C 180,E1 -9207.854,E2 -9207.854} C_VEL
LIN {X 0,Y 592.523,Z 341.946,A -85,B 0,C 180,E1 -9208.159,E2 -9208.159} C_VEL
LIN {X 0,Y 593.058,Z 318.859,A -85,B 0,C 180,E1 -9211.112,E2 -9211.112} C_VEL
LIN {X 0,Y 593.616,Z 295.76,A -85,B 0,C 180,E1 -9214.072,E2 -9214.072} C_VEL
LIN {X 0,Y 591.602,Z 283.924,A -85,B 0,C 180,E1 -9215.67,E2 -9215.67} C_VEL
LIN {X 0,Y 591.48,Z 283.369,A -85,B 0,C 180,E1 -9215.783,E2 -9215.783} C_VEL
LIN {X 0,Y 591.416,Z 283.374,A -85,B 0,C 180,E1 -9218.585,E2 -9218.585} C_VEL
LIN {X 0,Y 591.425,Z 283.371,A -85,B 0,C 180,E1 -9220.713,E2 -9220.713} C_VEL
LIN {X 0,Y 591.422,Z 283.371,A -85,B 0,C 180,E1 -9223.387,E2 -9223.387} C_VEL
LIN {X 0,Y 591.428,Z 283.373,A -85,B 0,C 180,E1 -9226.256,E2 -9226.256} C_VEL
LIN {X 0,Y 591.438,Z 283.37,A -85,B 0,C 180,E1 -9229.354,E2 -9229.354} C_VEL
LIN {X 0,Y 591.392,Z 283.378,A -85,B 0,C 180,E1 -9231.982,E2 -9231.982} C_VEL
LIN {X 0,Y 591.389,Z 283.376,A -85,B 0,C 180,E1 -9232.976,E2 -9232.976} C_VEL
LIN {X 0,Y 590.723,Z 283.461,A -85,B 0,C 180,E1 -9233.545,E2 -9233.545} C_VEL
LIN {X 0,Y 587.883,Z 283.815,A -85,B 0,C 180,E1 -9234.468,E2 -9234.468} C_VEL
LIN {X 0,Y 585.482,Z 284.115,A -85,B 0,C 180,E1 -9235.211,E2 -9235.211} C_VEL
LIN {X 0,Y 584.445,Z 284.243,A -85,B 0,C 180,E1 -9235.784,E2 -9235.784} C_VEL
LIN {X 0,Y 584.358,Z 284.253,A -85,B 0,C 180,E1 -9235.978,E2 -9235.978} C_VEL
LIN {X 0,Y 584.363,Z 284.252,A -85,B 0,C 180,E1 -9238.973,E2 -9238.973} C_VEL
LIN {X 0,Y 584.393,Z 284.249,A -85,B 0,C 180,E1 -9241.35,E2 -9241.35} C_VEL
LIN {X 0,Y 584.368,Z 284.25,A -85,B 0,C 180,E1 -9244.024,E2 -9244.024} C_VEL
LIN {X 0,Y 584.39,Z 284.249,A -85,B 0,C 180,E1 -9246.699,E2 -9246.699} C_VEL
LIN {X 0,Y 584.443,Z 284.242,A -85,B 0,C 180,E1 -9249.198,E2 -9249.198} C_VEL
LIN {X 0,Y 584.414,Z 284.245,A -85,B 0,C 180,E1 -9251.842,E2 -9251.842} C_VEL
LIN {X 0,Y 584.438,Z 284.244,A -85,B 0,C 180,E1 -9253.998,E2 -9253.998} C_VEL
LIN {X 0,Y 584.464,Z 284.237,A -85,B 0,C 180,E1 -9256.837,E2 -9256.837} C_VEL
LIN {X 0,Y 584.499,Z 284.235,A -85,B 0,C 180,E1 -9259.643,E2 -9259.643} C_VEL
LIN {X 0,Y 584.527,Z 284.234,A -85,B 0,C 180,E1 -9262.424,E2 -9262.424} C_VEL
LIN {X 0,Y 584.551,Z 284.302,A -85,B 0,C 180,E1 -9263.203,E2 -9263.203} C_VEL
LIN {X 0,Y 585.556,Z 291.489,A -85,B 0,C 180,E1 -9264.507,E2 -9264.507} C_VEL
LIN {X 0,Y 585.328,Z 298.914,A -85,B 0,C 180,E1 -9265.795,E2 -9265.795} C_VEL
LIN {X 0,Y 588.429,Z 314.195,A -85,B 0,C 180,E1 -9266.074,E2 -9266.074} C_VEL
LIN {X 0,Y 587.498,Z 434.747,A -85,B 0,C 180,E1 -9267.564,E2 -9267.564} C_VEL
LIN {X 0,Y 587.263,Z 449.04,A -85,B 0,C 180,E1 -9267.884,E2 -9267.884} C_VEL
LIN {X 0,Y 586.955,Z 462.772,A -85,B 0,C 180,E1 -9268.332,E2 -9268.332} C_VEL
LIN {X 0,Y 586.593,Z 475.57,A -85,B 0,C 180,E1 -9268.887,E2 -9268.887} C_VEL
LIN {X 0,Y 586.193,Z 487.995,A -85,B 0,C 180,E1 -9269.57,E2 -9269.57} C_VEL
LIN {X 0,Y 585.636,Z 499.392,A -85,B 0,C 180,E1 -9270.341,E2 -9270.341} C_VEL
LIN {X 0,Y 585.279,Z 509.811,A -85,B 0,C 180,E1 -9271.198,E2 -9271.198} C_VEL
LIN {X 0,Y 584.743,Z 520.214,A -85,B 0,C 180,E1 -9272.229,E2 -9272.229} C_VEL
LIN {X 0,Y 584.405,Z 528.791,A -85,B 0,C 180,E1 -9273.262,E2 -9273.262} C_VEL
LIN {X 0,Y 583.978,Z 537.06,A -85,B 0,C 180,E1 -9274.47,E2 -9274.47} C_VEL
LIN {X 0,Y 583.898,Z 542.795,A -85,B 0,C 180,E1 -9275.505,E2 -9275.505} C_VEL
LIN {X 0,Y 583.652,Z 548.97,A -85,B 0,C 180,E1 -9276.891,E2 -9276.891} C_VEL
LIN {X 0,Y 583.414,Z 553.506,A -85,B 0,C 180,E1 -9278.282,E2 -9278.282} C_VEL
LIN {X 0,Y 583.388,Z 556.573,A -85,B 0,C 180,E1 -9279.675,E2 -9279.675} C_VEL
LIN {X 0,Y 583.321,Z 558.28,A -85,B 0,C 180,E1 -9281.075,E2 -9281.075} C_VEL
LIN {X 0,Y 583.321,Z 558.637,A -85,B 0,C 180,E1 -9282.481,E2 -9282.481} C_VEL
LIN {X 0,Y 583.361,Z 557.638,A -85,B 0,C 180,E1 -9283.893,E2 -9283.893} C_VEL
LIN {X 0,Y 583.443,Z 555.247,A -85,B 0,C 180,E1 -9285.313,E2 -9285.313} C_VEL
LIN {X 0,Y 583.611,Z 551.374,A -85,B 0,C 180,E1 -9286.739,E2 -9286.739} C_VEL
LIN {X 0,Y 583.777,Z 547.359,A -85,B 0,C 180,E1 -9287.814,E2 -9287.814} C_VEL
LIN {X 0,Y 584.055,Z 542.356,A -85,B 0,C 180,E1 -9288.891,E2 -9288.891} C_VEL
LIN {X 0,Y 584.371,Z 535.078,A -85,B 0,C 180,E1 -9290.156,E2 -9290.156} C_VEL
LIN {X 0,Y 584.744,Z 527.371,A -85,B 0,C 180,E1 -9291.243,E2 -9291.243} C_VEL
LIN {X 0,Y 585.287,Z 518.024,A -85,B 0,C 180,E1 -9292.33,E2 -9292.33} C_VEL
LIN {X 0,Y 585.775,Z 507.591,A -85,B 0,C 180,E1 -9293.332,E2 -9293.332} C_VEL
LIN {X 0,Y 586.402,Z 496,A -85,B 0,C 180,E1 -9294.24,E2 -9294.24} C_VEL
LIN {X 0,Y 586.862,Z 483.795,A -85,B 0,C 180,E1 -9295.019,E2 -9295.019} C_VEL
LIN {X 0,Y 587.367,Z 470.173,A -85,B 0,C 180,E1 -9295.705,E2 -9295.705} C_VEL
LIN {X 0,Y 587.819,Z 456.453,A -85,B 0,C 180,E1 -9296.232,E2 -9296.232} C_VEL
LIN {X 0,Y 588.102,Z 442.407,A -85,B 0,C 180,E1 -9296.624,E2 -9296.624} C_VEL
LIN {X 0,Y 588.224,Z 427.842,A -85,B 0,C 180,E1 -9296.883,E2 -9296.883} C_VEL
LIN {X 0,Y 589.174,Z 314.094,A -85,B 0,C 180,E1 -9298.289,E2 -9298.289} C_VEL
LIN {X 0,Y 585.929,Z 299.399,A -85,B 0,C 180,E1 -9298.588,E2 -9298.588} C_VEL
LIN {X 0,Y 585.992,Z 292.977,A -85,B 0,C 180,E1 -9299.737,E2 -9299.737} C_VEL
LIN {X 0,Y 584.368,Z 284.255,A -85,B 0,C 180,E1 -9301.424,E2 -9301.424} C_VEL
LIN {X 0,Y 584.348,Z 284.256,A -85,B 0,C 180,E1 -9304.287,E2 -9304.287} C_VEL
LIN {X 0,Y 584.361,Z 284.25,A -85,B 0,C 180,E1 -9306.819,E2 -9306.819} C_VEL
LIN {X 0,Y 584.336,Z 284.252,A -85,B 0,C 180,E1 -9309.44,E2 -9309.44} C_VEL
LIN {X 0,Y 584.374,Z 284.251,A -85,B 0,C 180,E1 -9312.159,E2 -9312.159} C_VEL
LIN {X 0,Y 584.376,Z 284.238,A -85,B 0,C 180,E1 -9315.003,E2 -9315.003} C_VEL
LIN {X 0,Y 584.382,Z 284.251,A -85,B 0,C 180,E1 -9317.996,E2 -9317.996} C_VEL
LIN {X 0,Y 584.341,Z 284.251,A -85,B 0,C 180,E1 -9320.557,E2 -9320.557} C_VEL
LIN {X 0,Y 584.397,Z 284.244,A -85,B 0,C 180,E1 -9323.418,E2 -9323.418} C_VEL
LIN {X 0,Y 584.37,Z 284.246,A -85,B 0,C 180,E1 -9325.793,E2 -9325.793} C_VEL
LIN {X 0,Y 584.388,Z 284.242,A -85,B 0,C 180,E1 -9328.976,E2 -9328.976} C_VEL
LIN {X 0,Y 584.406,Z 284.247,A -85,B 0,C 180,E1 -9331.352,E2 -9331.352} C_VEL
LIN {X 0,Y 584.333,Z 284.251,A -85,B 0,C 180,E1 -9334.435,E2 -9334.435} C_VEL
LIN {X 0,Y 584.375,Z 284.241,A -85,B 0,C 180,E1 -9336.7,E2 -9336.7} C_VEL
LIN {X 0,Y 584.413,Z 284.246,A -85,B 0,C 180,E1 -9339.199,E2 -9339.199} C_VEL
LIN {X 0,Y 584.374,Z 284.249,A -85,B 0,C 180,E1 -9341.842,E2 -9341.842} C_VEL
LIN {X 0,Y 584.42,Z 284.24,A -85,B 0,C 180,E1 -9344.712,E2 -9344.712} C_VEL
LIN {X 0,Y 584.447,Z 284.233,A -85,B 0,C 180,E1 -9346.838,E2 -9346.838} C_VEL
LIN {X 0,Y 584.453,Z 284.236,A -85,B 0,C 180,E1 -9349.644,E2 -9349.644} C_VEL
LIN {X 0,Y 584.503,Z 284.227,A -85,B 0,C 180,E1 -9352.425,E2 -9352.425} C_VEL
LIN {X 0,Y 584.562,Z 284.226,A -85,B 0,C 180,E1 -9355.189,E2 -9355.189} C_VEL
LIN {X 0,Y 584.688,Z 284.212,A -85,B 0,C 180,E1 -9359.314,E2 -9359.314} C_VEL
LIN {X 0,Y 584.645,Z 284.209,A -85,B 0,C 180,E1 -9361.373,E2 -9361.373} C_VEL
LIN {X 0,Y 584.576,Z 284.226,A -85,B 0,C 180,E1 -9364.811,E2 -9364.811} C_VEL
LIN {X 0,Y 584.504,Z 284.225,A -85,B 0,C 180,E1 -9367.575,E2 -9367.575} C_VEL
LIN {X 0,Y 584.542,Z 284.23,A -85,B 0,C 180,E1 -9370.721,E2 -9370.721} C_VEL
LIN {X 0,Y 584.458,Z 284.232,A -85,B 0,C 180,E1 -9373.904,E2 -9373.904} C_VEL
LIN {X 0,Y 584.441,Z 284.24,A -85,B 0,C 180,E1 -9376.717,E2 -9376.717} C_VEL
LIN {X 0,Y 584.38,Z 284.244,A -85,B 0,C 180,E1 -9379.61,E2 -9379.61} C_VEL
LIN {X 0,Y 584.42,Z 284.235,A -85,B 0,C 180,E1 -9381.811,E2 -9381.811} C_VEL
LIN {X 0,Y 584.369,Z 284.251,A -85,B 0,C 180,E1 -9384.804,E2 -9384.804} C_VEL
LIN {X 0,Y 584.379,Z 284.245,A -85,B 0,C 180,E1 -9387.87,E2 -9387.87} C_VEL
LIN {X 0,Y 584.382,Z 284.249,A -85,B 0,C 180,E1 -9390.35,E2 -9390.35} C_VEL
LIN {X 0,Y 584.383,Z 284.245,A -85,B 0,C 180,E1 -9392.967,E2 -9392.967} C_VEL
LIN {X 0,Y 584.413,Z 284.228,A -85,B 0,C 180,E1 -9395.965,E2 -9395.965} C_VEL
LIN {X 0,Y 584.394,Z 284.246,A -85,B 0,C 180,E1 -9398.828,E2 -9398.828} C_VEL
LIN {X 0,Y 584.366,Z 284.247,A -85,B 0,C 180,E1 -9401.243,E2 -9401.243} C_VEL
LIN {X 0,Y 584.378,Z 284.251,A -85,B 0,C 180,E1 -9404.043,E2 -9404.043} C_VEL
LIN {X 0,Y 584.394,Z 284.243,A -85,B 0,C 180,E1 -9406.982,E2 -9406.982} C_VEL
LIN {X 0,Y 584.401,Z 284.245,A -85,B 0,C 180,E1 -9409.67,E2 -9409.67} C_VEL
LIN {X 0,Y 584.42,Z 284.246,A -85,B 0,C 180,E1 -9412.323,E2 -9412.323} C_VEL
LIN {X 0,Y 584.427,Z 284.245,A -85,B 0,C 180,E1 -9414.883,E2 -9414.883} C_VEL
LIN {X 0,Y 584.379,Z 284.252,A -85,B 0,C 180,E1 -9417.361,E2 -9417.361} C_VEL
LIN {X 0,Y 584.404,Z 284.254,A -85,B 0,C 180,E1 -9419.778,E2 -9419.778} C_VEL
LIN {X 0,Y 584.389,Z 284.251,A -85,B 0,C 180,E1 -9422.494,E2 -9422.494} C_VEL
LIN {X 0,Y 584.411,Z 284.445,A -85,B 0,C 180,E1 -9423.246,E2 -9423.246} C_VEL
LIN {X 0,Y 587.544,Z 298.971,A -85,B 0,C 180,E1 -9425.341,E2 -9425.341} C_VEL
LIN {X 0,Y 587.849,Z 303.218,A -85,B 0,C 180,E1 -9425.917,E2 -9425.917} C_VEL
LIN {X 0,Y 586.762,Z 324.939,A -85,B 0,C 180,E1 -9428.713,E2 -9428.713} C_VEL
LIN {X 0,Y 585.803,Z 347.147,A -85,B 0,C 180,E1 -9431.529,E2 -9431.529} C_VEL
LIN {X 0,Y 585.214,Z 362.45,A -85,B 0,C 180,E1 -9433.431,E2 -9433.431} C_VEL
LIN {X 0,Y 588.486,Z 385.423,A -85,B 0,C 180,E1 -9433.826,E2 -9433.826} C_VEL
LIN {X 0,Y 588.799,Z 392.392,A -85,B 0,C 180,E1 -9433.923,E2 -9433.923} C_VEL
LIN {X 0,Y 587.862,Z 500.569,A -85,B 0,C 180,E1 -9435.272,E2 -9435.272} C_VEL
LIN {X 0,Y 587.415,Z 515.034,A -85,B 0,C 180,E1 -9435.589,E2 -9435.589} C_VEL
LIN {X 0,Y 586.912,Z 528.429,A -85,B 0,C 180,E1 -9436.017,E2 -9436.017} C_VEL
LIN {X 0,Y 586.347,Z 542.436,A -85,B 0,C 180,E1 -9436.619,E2 -9436.619} C_VEL
LIN {X 0,Y 585.722,Z 554.971,A -85,B 0,C 180,E1 -9437.308,E2 -9437.308} C_VEL
LIN {X 0,Y 585.178,Z 566.43,A -85,B 0,C 180,E1 -9438.086,E2 -9438.086} C_VEL
LIN {X 0,Y 584.677,Z 576.98,A -85,B 0,C 180,E1 -9438.951,E2 -9438.951} C_VEL
LIN {X 0,Y 584.339,Z 585.856,A -85,B 0,C 180,E1 -9439.818,E2 -9439.818} C_VEL
LIN {X 0,Y 583.915,Z 594.818,A -85,B 0,C 180,E1 -9440.856,E2 -9440.856} C_VEL
LIN {X 0,Y 583.601,Z 603.426,A -85,B 0,C 180,E1 -9442.068,E2 -9442.068} C_VEL
LIN {X 0,Y 583.42,Z 611.651,A -85,B 0,C 180,E1 -9443.453,E2 -9443.453} C_VEL
LIN {X 0,Y 583.319,Z 616.721,A -85,B 0,C 180,E1 -9444.489,E2 -9444.489} C_VEL
LIN {X 0,Y 583.271,Z 621.908,A -85,B 0,C 180,E1 -9445.87,E2 -9445.87} C_VEL
LIN {X 0,Y 583.257,Z 625.529,A -85,B 0,C 180,E1 -9447.248,E2 -9447.248} C_VEL
LIN {X 0,Y 583.244,Z 627.691,A -85,B 0,C 180,E1 -9448.625,E2 -9448.625} C_VEL
LIN {X 0,Y 583.278,Z 628.445,A -85,B 0,C 180,E1 -9450.002,E2 -9450.002} C_VEL
LIN {X 0,Y 583.243,Z 627.788,A -85,B 0,C 180,E1 -9451.378,E2 -9451.378} C_VEL
LIN {X 0,Y 583.259,Z 625.702,A -85,B 0,C 180,E1 -9452.755,E2 -9452.755} C_VEL
LIN {X 0,Y 583.273,Z 622.159,A -85,B 0,C 180,E1 -9454.134,E2 -9454.134} C_VEL
LIN {X 0,Y 583.326,Z 617.055,A -85,B 0,C 180,E1 -9455.514,E2 -9455.514} C_VEL
LIN {X 0,Y 583.427,Z 612.097,A -85,B 0,C 180,E1 -9456.551,E2 -9456.551} C_VEL
LIN {X 0,Y 583.592,Z 604.927,A -85,B 0,C 180,E1 -9457.762,E2 -9457.762} C_VEL
LIN {X 0,Y 583.888,Z 596.037,A -85,B 0,C 180,E1 -9458.973,E2 -9458.973} C_VEL
LIN {X 0,Y 584.204,Z 586.709,A -85,B 0,C 180,E1 -9460.013,E2 -9460.013} C_VEL
LIN {X 0,Y 584.574,Z 576.473,A -85,B 0,C 180,E1 -9460.958,E2 -9460.958} C_VEL
LIN {X 0,Y 585.073,Z 562.699,A -85,B 0,C 180,E1 -9462.007,E2 -9462.007} C_VEL
LIN {X 0,Y 585.649,Z 550.179,A -85,B 0,C 180,E1 -9462.785,E2 -9462.785} C_VEL
LIN {X 0,Y 586.161,Z 538.126,A -85,B 0,C 180,E1 -9463.388,E2 -9463.388} C_VEL
LIN {X 0,Y 586.588,Z 524.91,A -85,B 0,C 180,E1 -9463.906,E2 -9463.906} C_VEL
LIN {X 0,Y 587.035,Z 510.612,A -85,B 0,C 180,E1 -9464.314,E2 -9464.314} C_VEL
LIN {X 0,Y 587.356,Z 495.973,A -85,B 0,C 180,E1 -9464.584,E2 -9464.584} C_VEL
LIN {X 0,Y 588.147,Z 398.964,A -85,B 0,C 180,E1 -9465.788,E2 -9465.788} C_VEL
LIN {X 0,Y 588.164,Z 387.059,A -85,B 0,C 180,E1 -9465.965,E2 -9465.965} C_VEL
LIN {X 0,Y 585.098,Z 361.631,A -85,B 0,C 180,E1 -9466.453,E2 -9466.453} C_VEL
LIN {X 0,Y 585.952,Z 334.809,A -85,B 0,C 180,E1 -9469.738,E2 -9469.738} C_VEL
LIN {X 0,Y 586.861,Z 311.53,A -85,B 0,C 180,E1 -9472.64,E2 -9472.64} C_VEL
LIN {X 0,Y 587.241,Z 298.401,A -85,B 0,C 180,E1 -9474.301,E2 -9474.301} C_VEL
LIN {X 0,Y 584.383,Z 284.253,A -85,B 0,C 180,E1 -9476.23,E2 -9476.23} C_VEL
LIN {X 0,Y 584.391,Z 284.247,A -85,B 0,C 180,E1 -9478.958,E2 -9478.958} C_VEL
LIN {X 0,Y 584.385,Z 284.25,A -85,B 0,C 180,E1 -9481.83,E2 -9481.83} C_VEL
LIN {X 0,Y 584.365,Z 284.251,A -85,B 0,C 180,E1 -9484.29,E2 -9484.29} C_VEL
LIN {X 0,Y 584.371,Z 284.249,A -85,B 0,C 180,E1 -9486.822,E2 -9486.822} C_VEL
LIN {X 0,Y 584.355,Z 284.256,A -85,B 0,C 180,E1 -9489.443,E2 -9489.443} C_VEL
LIN {X 0,Y 584.354,Z 284.248,A -85,B 0,C 180,E1 -9492.165,E2 -9492.165} C_VEL
LIN {X 0,Y 584.379,Z 284.252,A -85,B 0,C 180,E1 -9495.007,E2 -9495.007} C_VEL
LIN {X 0,Y 584.354,Z 284.25,A -85,B 0,C 180,E1 -9497.836,E2 -9497.836} C_VEL
LIN {X 0,Y 584.355,Z 284.253,A -85,B 0,C 180,E1 -9500.558,E2 -9500.558} C_VEL
LIN {X 0,Y 584.4,Z 284.246,A -85,B 0,C 180,E1 -9503.423,E2 -9503.423} C_VEL
LIN {X 0,Y 584.374,Z 284.247,A -85,B 0,C 180,E1 -9505.798,E2 -9505.798} C_VEL
LIN {X 0,Y 584.401,Z 284.249,A -85,B 0,C 180,E1 -9508.32,E2 -9508.32} C_VEL
LIN {X 0,Y 584.396,Z 284.244,A -85,B 0,C 180,E1 -9511.352,E2 -9511.352} C_VEL
LIN {X 0,Y 584.367,Z 284.254,A -85,B 0,C 180,E1 -9514.026,E2 -9514.026} C_VEL
LIN {X 0,Y 584.392,Z 284.251,A -85,B 0,C 180,E1 -9516.701,E2 -9516.701} C_VEL
LIN {X 0,Y 584.445,Z 284.244,A -85,B 0,C 180,E1 -9519.2,E2 -9519.2} C_VEL
LIN {X 0,Y 584.399,Z 284.254,A -85,B 0,C 180,E1 -9521.843,E2 -9521.843} C_VEL
LIN {X 0,Y 584.436,Z 284.243,A -85,B 0,C 180,E1 -9524.712,E2 -9524.712} C_VEL
LIN {X 0,Y 584.464,Z 284.242,A -85,B 0,C 180,E1 -9526.838,E2 -9526.838} C_VEL
LIN {X 0,Y 584.451,Z 284.281,A -85,B 0,C 180,E1 -9527.981,E2 -9527.981} C_VEL
LIN {X 0,Y 586.983,Z 296.937,A -85,B 0,C 180,E1 -9529.689,E2 -9529.689} C_VEL
LIN {X 0,Y 586.69,Z 317.449,A -85,B 0,C 180,E1 -9532.282,E2 -9532.282} C_VEL
LIN {X 0,Y 585.985,Z 342.807,A -85,B 0,C 180,E1 -9535.479,E2 -9535.479} C_VEL
LIN {X 0,Y 588.963,Z 359.778,A -85,B 0,C 180,E1 -9535.844,E2 -9535.844} C_VEL
LIN {X 0,Y 587.443,Z 481.297,A -85,B 0,C 180,E1 -9537.565,E2 -9537.565} C_VEL
LIN {X 0,Y 587.126,Z 495.857,A -85,B 0,C 180,E1 -9537.906,E2 -9537.906} C_VEL
LIN {X 0,Y 586.668,Z 509.726,A -85,B 0,C 180,E1 -9538.375,E2 -9538.375} C_VEL
LIN {X 0,Y 586.203,Z 523.052,A -85,B 0,C 180,E1 -9538.973,E2 -9538.973} C_VEL
LIN {X 0,Y 585.692,Z 535.178,A -85,B 0,C 180,E1 -9539.657,E2 -9539.657} C_VEL
LIN {X 0,Y 585.3,Z 547.429,A -85,B 0,C 180,E1 -9540.514,E2 -9540.514} C_VEL
LIN {X 0,Y 584.825,Z 557.59,A -85,B 0,C 180,E1 -9541.373,E2 -9541.373} C_VEL
LIN {X 0,Y 584.307,Z 567.764,A -85,B 0,C 180,E1 -9542.405,E2 -9542.405} C_VEL
LIN {X 0,Y 584.008,Z 576.161,A -85,B 0,C 180,E1 -9543.438,E2 -9543.438} C_VEL
LIN {X 0,Y 583.763,Z 583.154,A -85,B 0,C 180,E1 -9544.473,E2 -9544.473} C_VEL
LIN {X 0,Y 583.569,Z 590.034,A -85,B 0,C 180,E1 -9545.727,E2 -9545.727} C_VEL
LIN {X 0,Y 583.409,Z 595.165,A -85,B 0,C 180,E1 -9546.896,E2 -9546.896} C_VEL
LIN {X 0,Y 583.235,Z 599.689,A -85,B 0,C 180,E1 -9548.286,E2 -9548.286} C_VEL
LIN {X 0,Y 583.242,Z 602.705,A -85,B 0,C 180,E1 -9549.679,E2 -9549.679} C_VEL
LIN {X 0,Y 583.13,Z 604.305,A -85,B 0,C 180,E1 -9551.081,E2 -9551.081} C_VEL
LIN {X 0,Y 583.158,Z 604.489,A -85,B 0,C 180,E1 -9552.486,E2 -9552.486} C_VEL
LIN {X 0,Y 583.18,Z 603.242,A -85,B 0,C 180,E1 -9553.899,E2 -9553.899} C_VEL
LIN {X 0,Y 583.207,Z 600.476,A -85,B 0,C 180,E1 -9555.321,E2 -9555.321} C_VEL
LIN {X 0,Y 583.295,Z 597.51,A -85,B 0,C 180,E1 -9556.356,E2 -9556.356} C_VEL
LIN {X 0,Y 583.368,Z 593.32,A -85,B 0,C 180,E1 -9557.468,E2 -9557.468} C_VEL
LIN {X 0,Y 583.545,Z 587.734,A -85,B 0,C 180,E1 -9558.638,E2 -9558.638} C_VEL
LIN {X 0,Y 583.779,Z 580.748,A -85,B 0,C 180,E1 -9559.813,E2 -9559.813} C_VEL
LIN {X 0,Y 584.058,Z 573.284,A -85,B 0,C 180,E1 -9560.844,E2 -9560.844} C_VEL
LIN {X 0,Y 584.322,Z 564.901,A -85,B 0,C 180,E1 -9561.815,E2 -9561.815} C_VEL
LIN {X 0,Y 584.768,Z 554.842,A -85,B 0,C 180,E1 -9562.788,E2 -9562.788} C_VEL
LIN {X 0,Y 585.148,Z 544.232,A -85,B 0,C 180,E1 -9563.641,E2 -9563.641} C_VEL
LIN {X 0,Y 585.655,Z 531.981,A -85,B 0,C 180,E1 -9564.451,E2 -9564.451} C_VEL
LIN {X 0,Y 586.04,Z 518.683,A -85,B 0,C 180,E1 -9565.154,E2 -9565.154} C_VEL
LIN {X 0,Y 586.493,Z 505.366,A -85,B 0,C 180,E1 -9565.701,E2 -9565.701} C_VEL
LIN {X 0,Y 586.863,Z 491.182,A -85,B 0,C 180,E1 -9566.135,E2 -9566.135} C_VEL
LIN {X 0,Y 587.095,Z 476.295,A -85,B 0,C 180,E1 -9566.441,E2 -9566.441} C_VEL
LIN {X 0,Y 588.324,Z 359.748,A -85,B 0,C 180,E1 -9568.008,E2 -9568.008} C_VEL
LIN {X 0,Y 585.54,Z 342.024,A -85,B 0,C 180,E1 -9568.335,E2 -9568.335} C_VEL
LIN {X 0,Y 586.078,Z 320.365,A -85,B 0,C 180,E1 -9571.124,E2 -9571.124} C_VEL
LIN {X 0,Y 586.686,Z 297.034,A -85,B 0,C 180,E1 -9574.134,E2 -9574.134} C_VEL
LIN {X 0,Y 584.455,Z 284.244,A -85,B 0,C 180,E1 -9575.896,E2 -9575.896} C_VEL
LIN {X 0,Y 584.367,Z 284.249,A -85,B 0,C 180,E1 -9578.819,E2 -9578.819} C_VEL
LIN {X 0,Y 584.35,Z 284.251,A -85,B 0,C 180,E1 -9581.244,E2 -9581.244} C_VEL
LIN {X 0,Y 584.4,Z 284.25,A -85,B 0,C 180,E1 -9584.041,E2 -9584.041} C_VEL
LIN {X 0,Y 584.364,Z 284.25,A -85,B 0,C 180,E1 -9586.985,E2 -9586.985} C_VEL
LIN {X 0,Y 584.361,Z 284.253,A -85,B 0,C 180,E1 -9590.097,E2 -9590.097} C_VEL
LIN {X 0,Y 584.345,Z 284.252,A -85,B 0,C 180,E1 -9592.978,E2 -9592.978} C_VEL
LIN {X 0,Y 584.365,Z 284.254,A -85,B 0,C 180,E1 -9595.71,E2 -9595.71} C_VEL
LIN {X 0,Y 584.358,Z 284.253,A -85,B 0,C 180,E1 -9595.978,E2 -9595.978} C_VEL
LIN {X 0,Y 583.683,Z 284.337,A -85,B 0,C 180,E1 -9596.553,E2 -9596.553} C_VEL
LIN {X 0,Y 580.826,Z 284.693,A -85,B 0,C 180,E1 -9597.487,E2 -9597.487} C_VEL
LIN {X 0,Y 578.419,Z 284.992,A -85,B 0,C 180,E1 -9598.239,E2 -9598.239} C_VEL
LIN {X 0,Y 577.389,Z 285.122,A -85,B 0,C 180,E1 -9598.819,E2 -9598.819} C_VEL
LIN {X 0,Y 577.307,Z 285.13,A -85,B 0,C 180,E1 -9599.015,E2 -9599.015} C_VEL
LIN {X 0,Y 577.333,Z 285.127,A -85,B 0,C 180,E1 -9601.759,E2 -9601.759} C_VEL
LIN {X 0,Y 577.322,Z 285.128,A -85,B 0,C 180,E1 -9604.1,E2 -9604.1} C_VEL
LIN {X 0,Y 577.361,Z 285.127,A -85,B 0,C 180,E1 -9606.398,E2 -9606.398} C_VEL
LIN {X 0,Y 577.401,Z 285.118,A -85,B 0,C 180,E1 -9609.081,E2 -9609.081} C_VEL
LIN {X 0,Y 577.39,Z 285.119,A -85,B 0,C 180,E1 -9611.613,E2 -9611.613} C_VEL
LIN {X 0,Y 577.416,Z 285.117,A -85,B 0,C 180,E1 -9614.52,E2 -9614.52} C_VEL
LIN {X 0,Y 577.417,Z 285.115,A -85,B 0,C 180,E1 -9616.673,E2 -9616.673} C_VEL
LIN {X 0,Y 577.454,Z 285.111,A -85,B 0,C 180,E1 -9619.515,E2 -9619.515} C_VEL
LIN {X 0,Y 577.481,Z 285.112,A -85,B 0,C 180,E1 -9622.331,E2 -9622.331} C_VEL
LIN {X 0,Y 577.502,Z 285.216,A -85,B 0,C 180,E1 -9623.098,E2 -9623.098} C_VEL
LIN {X 0,Y 578.561,Z 292.552,A -85,B 0,C 180,E1 -9624.44,E2 -9624.44} C_VEL
LIN {X 0,Y 578.371,Z 299.245,A -85,B 0,C 180,E1 -9625.614,E2 -9625.614} C_VEL
LIN {X 0,Y 581.604,Z 315.711,A -85,B 0,C 180,E1 -9625.919,E2 -9625.919} C_VEL
LIN {X 0,Y 580.606,Z 434.77,A -85,B 0,C 180,E1 -9627.405,E2 -9627.405} C_VEL
LIN {X 0,Y 580.356,Z 449.195,A -85,B 0,C 180,E1 -9627.729,E2 -9627.729} C_VEL
LIN {X 0,Y 580.031,Z 462.993,A -85,B 0,C 180,E1 -9628.182,E2 -9628.182} C_VEL
LIN {X 0,Y 579.642,Z 476.697,A -85,B 0,C 180,E1 -9628.787,E2 -9628.787} C_VEL
LIN {X 0,Y 579.2,Z 489,A -85,B 0,C 180,E1 -9629.479,E2 -9629.479} C_VEL
LIN {X 0,Y 578.597,Z 501.449,A -85,B 0,C 180,E1 -9630.345,E2 -9630.345} C_VEL
LIN {X 0,Y 578.234,Z 511.594,A -85,B 0,C 180,E1 -9631.213,E2 -9631.213} C_VEL
LIN {X 0,Y 577.675,Z 521.761,A -85,B 0,C 180,E1 -9632.257,E2 -9632.257} C_VEL
LIN {X 0,Y 577.345,Z 530.152,A -85,B 0,C 180,E1 -9633.302,E2 -9633.302} C_VEL
LIN {X 0,Y 576.911,Z 538.205,A -85,B 0,C 180,E1 -9634.525,E2 -9634.525} C_VEL
LIN {X 0,Y 576.82,Z 543.855,A -85,B 0,C 180,E1 -9635.573,E2 -9635.573} C_VEL
LIN {X 0,Y 576.606,Z 548.482,A -85,B 0,C 180,E1 -9636.625,E2 -9636.625} C_VEL
LIN {X 0,Y 576.364,Z 553.293,A -85,B 0,C 180,E1 -9638.032,E2 -9638.032} C_VEL
LIN {X 0,Y 576.333,Z 555.887,A -85,B 0,C 180,E1 -9639.089,E2 -9639.089} C_VEL
LIN {X 0,Y 576.255,Z 558.156,A -85,B 0,C 180,E1 -9640.503,E2 -9640.503} C_VEL
LIN {X 0,Y 576.201,Z 559.074,A -85,B 0,C 180,E1 -9641.925,E2 -9641.925} C_VEL
LIN {X 0,Y 576.3,Z 558.636,A -85,B 0,C 180,E1 -9643.35,E2 -9643.35} C_VEL
LIN {X 0,Y 576.33,Z 556.832,A -85,B 0,C 180,E1 -9644.785,E2 -9644.785} C_VEL
LIN {X 0,Y 576.516,Z 553.566,A -85,B 0,C 180,E1 -9646.225,E2 -9646.225} C_VEL
LIN {X 0,Y 576.688,Z 548.703,A -85,B 0,C 180,E1 -9647.675,E2 -9647.675} C_VEL
LIN {X 0,Y 576.972,Z 544.02,A -85,B 0,C 180,E1 -9648.752,E2 -9648.752} C_VEL
LIN {X 0,Y 577.298,Z 536.965,A -85,B 0,C 180,E1 -9650.043,E2 -9650.043} C_VEL
LIN {X 0,Y 577.67,Z 529.851,A -85,B 0,C 180,E1 -9651.107,E2 -9651.107} C_VEL
LIN {X 0,Y 578.224,Z 520.605,A -85,B 0,C 180,E1 -9652.242,E2 -9652.242} C_VEL
LIN {X 0,Y 578.76,Z 510.898,A -85,B 0,C 180,E1 -9653.228,E2 -9653.228} C_VEL
LIN {X 0,Y 579.363,Z 499.593,A -85,B 0,C 180,E1 -9654.174,E2 -9654.174} C_VEL
LIN {X 0,Y 579.903,Z 487.419,A -85,B 0,C 180,E1 -9655.006,E2 -9655.006} C_VEL
LIN {X 0,Y 580.385,Z 475.688,A -85,B 0,C 180,E1 -9655.653,E2 -9655.653} C_VEL
LIN {X 0,Y 580.851,Z 463,A -85,B 0,C 180,E1 -9656.207,E2 -9656.207} C_VEL
LIN {X 0,Y 581.21,Z 448.948,A -85,B 0,C 180,E1 -9656.669,E2 -9656.669} C_VEL
LIN {X 0,Y 581.416,Z 435.038,A -85,B 0,C 180,E1 -9656.982,E2 -9656.982} C_VEL
LIN {X 0,Y 582.522,Z 315.544,A -85,B 0,C 180,E1 -9658.492,E2 -9658.492} C_VEL
LIN {X 0,Y 579.012,Z 299.681,A -85,B 0,C 180,E1 -9658.837,E2 -9658.837} C_VEL
LIN {X 0,Y 578.943,Z 293.631,A -85,B 0,C 180,E1 -9659.936,E2 -9659.936} C_VEL
LIN {X 0,Y 577.325,Z 285.132,A -85,B 0,C 180,E1 -9661.593,E2 -9661.593} C_VEL
LIN {X 0,Y 577.313,Z 285.131,A -85,B 0,C 180,E1 -9664.408,E2 -9664.408} C_VEL
LIN {X 0,Y 577.329,Z 285.126,A -85,B 0,C 180,E1 -9666.799,E2 -9666.799} C_VEL
LIN {X 0,Y 577.303,Z 285.135,A -85,B 0,C 180,E1 -9670.017,E2 -9670.017} C_VEL
LIN {X 0,Y 577.323,Z 285.127,A -85,B 0,C 180,E1 -9672.796,E2 -9672.796} C_VEL
LIN {X 0,Y 577.342,Z 285.12,A -85,B 0,C 180,E1 -9675.706,E2 -9675.706} C_VEL
LIN {X 0,Y 577.326,Z 285.131,A -85,B 0,C 180,E1 -9678.142,E2 -9678.142} C_VEL
LIN {X 0,Y 577.296,Z 285.128,A -85,B 0,C 180,E1 -9680.881,E2 -9680.881} C_VEL
LIN {X 0,Y 577.347,Z 285.119,A -85,B 0,C 180,E1 -9683.525,E2 -9683.525} C_VEL
LIN {X 0,Y 577.31,Z 285.131,A -85,B 0,C 180,E1 -9686.075,E2 -9686.075} C_VEL
LIN {X 0,Y 577.328,Z 285.121,A -85,B 0,C 180,E1 -9688.554,E2 -9688.554} C_VEL
LIN {X 0,Y 577.366,Z 285.12,A -85,B 0,C 180,E1 -9690.97,E2 -9690.97} C_VEL
LIN {X 0,Y 577.29,Z 285.135,A -85,B 0,C 180,E1 -9693.873,E2 -9693.873} C_VEL
LIN {X 0,Y 577.347,Z 285.116,A -85,B 0,C 180,E1 -9696.399,E2 -9696.399} C_VEL
LIN {X 0,Y 577.367,Z 285.127,A -85,B 0,C 180,E1 -9699.401,E2 -9699.401} C_VEL
LIN {X 0,Y 577.317,Z 285.124,A -85,B 0,C 180,E1 -9702.343,E2 -9702.343} C_VEL
LIN {X 0,Y 577.405,Z 285.118,A -85,B 0,C 180,E1 -9705.241,E2 -9705.241} C_VEL
LIN {X 0,Y 577.404,Z 285.119,A -85,B 0,C 180,E1 -9707.387,E2 -9707.387} C_VEL
LIN {X 0,Y 577.411,Z 285.109,A -85,B 0,C 180,E1 -9710.222,E2 -9710.222} C_VEL
LIN {X 0,Y 577.472,Z 285.109,A -85,B 0,C 180,E1 -9713.033,E2 -9713.033} C_VEL
LIN {X 0,Y 577.512,Z 285.094,A -85,B 0,C 180,E1 -9715.827,E2 -9715.827} C_VEL
LIN {X 0,Y 577.662,Z 285.088,A -85,B 0,C 180,E1 -9719.305,E2 -9719.305} C_VEL
LIN {X 0,Y 577.591,Z 285.087,A -85,B 0,C 180,E1 -9721.39,E2 -9721.39} C_VEL
LIN {X 0,Y 577.548,Z 285.103,A -85,B 0,C 180,E1 -9724.87,E2 -9724.87} C_VEL
LIN {X 0,Y 577.457,Z 285.102,A -85,B 0,C 180,E1 -9727.668,E2 -9727.668} C_VEL
LIN {X 0,Y 577.489,Z 285.11,A -85,B 0,C 180,E1 -9730.761,E2 -9730.761} C_VEL
LIN {X 0,Y 577.404,Z 285.111,A -85,B 0,C 180,E1 -9734.041,E2 -9734.041} C_VEL
LIN {X 0,Y 577.395,Z 285.114,A -85,B 0,C 180,E1 -9736.927,E2 -9736.927} C_VEL
LIN {X 0,Y 577.364,Z 285.122,A -85,B 0,C 180,E1 -9739.121,E2 -9739.121} C_VEL
LIN {X 0,Y 577.37,Z 285.114,A -85,B 0,C 180,E1 -9741.343,E2 -9741.343} C_VEL
LIN {X 0,Y 577.37,Z 285.123,A -85,B 0,C 180,E1 -9744.361,E2 -9744.361} C_VEL
LIN {X 0,Y 577.345,Z 285.12,A -85,B 0,C 180,E1 -9747.674,E2 -9747.674} C_VEL
LIN {X 0,Y 577.346,Z 285.121,A -85,B 0,C 180,E1 -9749.829,E2 -9749.829} C_VEL
LIN {X 0,Y 577.326,Z 285.129,A -85,B 0,C 180,E1 -9752.265,E2 -9752.265} C_VEL
LIN {X 0,Y 577.357,Z 285.109,A -85,B 0,C 180,E1 -9754.764,E2 -9754.764} C_VEL
LIN {X 0,Y 577.372,Z 285.114,A -85,B 0,C 180,E1 -9757.343,E2 -9757.343} C_VEL
LIN {X 0,Y 577.361,Z 285.125,A -85,B 0,C 180,E1 -9760.159,E2 -9760.159} C_VEL
LIN {X 0,Y 577.331,Z 285.125,A -85,B 0,C 180,E1 -9762.798,E2 -9762.798} C_VEL
LIN {X 0,Y 577.346,Z 285.122,A -85,B 0,C 180,E1 -9765.709,E2 -9765.709} C_VEL
LIN {X 0,Y 577.351,Z 285.129,A -85,B 0,C 180,E1 -9768.147,E2 -9768.147} C_VEL
LIN {X 0,Y 577.351,Z 285.121,A -85,B 0,C 180,E1 -9770.937,E2 -9770.937} C_VEL
LIN {X 0,Y 577.379,Z 285.119,A -85,B 0,C 180,E1 -9773.53,E2 -9773.53} C_VEL
LIN {X 0,Y 577.332,Z 285.13,A -85,B 0,C 180,E1 -9776.079,E2 -9776.079} C_VEL
LIN {X 0,Y 577.342,Z 285.13,A -85,B 0,C 180,E1 -9778.557,E2 -9778.557} C_VEL
LIN {X 0,Y 577.378,Z 285.122,A -85,B 0,C 180,E1 -9780.973,E2 -9780.973} C_VEL
LIN {X 0,Y 577.374,Z 285.249,A -85,B 0,C 180,E1 -9783.015,E2 -9783.015} C_VEL
LIN {X 0,Y 580.631,Z 300.259,A -85,B 0,C 180,E1 -9785.218,E2 -9785.218} C_VEL
LIN {X 0,Y 580.97,Z 304.507,A -85,B 0,C 180,E1 -9785.802,E2 -9785.802} C_VEL
LIN {X 0,Y 579.855,Z 325.637,A -85,B 0,C 180,E1 -9788.559,E2 -9788.559} C_VEL
LIN {X 0,Y 578.86,Z 346.964,A -85,B 0,C 180,E1 -9791.299,E2 -9791.299} C_VEL
LIN {X 0,Y 578.288,Z 361.88,A -85,B 0,C 180,E1 -9793.196,E2 -9793.196} C_VEL
LIN {X 0,Y 581.799,Z 386.825,A -85,B 0,C 180,E1 -9793.633,E2 -9793.633} C_VEL
LIN {X 0,Y 582.017,Z 396.134,A -85,B 0,C 180,E1 -9793.759,E2 -9793.759} C_VEL
LIN {X 0,Y 581.07,Z 499.831,A -85,B 0,C 180,E1 -9795.066,E2 -9795.066} C_VEL
LIN {X 0,Y 580.623,Z 513.918,A -85,B 0,C 180,E1 -9795.372,E2 -9795.372} C_VEL
LIN {X 0,Y 580.127,Z 527.49,A -85,B 0,C 180,E1 -9795.805,E2 -9795.805} C_VEL
LIN {X 0,Y 579.504,Z 540.723,A -85,B 0,C 180,E1 -9796.369,E2 -9796.369} C_VEL
LIN {X 0,Y 578.877,Z 553.498,A -85,B 0,C 180,E1 -9797.067,E2 -9797.067} C_VEL
LIN {X 0,Y 578.2,Z 566.307,A -85,B 0,C 180,E1 -9797.94,E2 -9797.94} C_VEL
LIN {X 0,Y 577.685,Z 576.801,A -85,B 0,C 180,E1 -9798.816,E2 -9798.816} C_VEL
LIN {X 0,Y 577.342,Z 585.632,A -85,B 0,C 180,E1 -9799.693,E2 -9799.693} C_VEL
LIN {X 0,Y 576.888,Z 594.56,A -85,B 0,C 180,E1 -9800.744,E2 -9800.744} C_VEL
LIN {X 0,Y 576.512,Z 603.138,A -85,B 0,C 180,E1 -9801.97,E2 -9801.97} C_VEL
LIN {X 0,Y 576.327,Z 611.357,A -85,B 0,C 180,E1 -9803.372,E2 -9803.372} C_VEL
LIN {X 0,Y 576.237,Z 616.465,A -85,B 0,C 180,E1 -9804.421,E2 -9804.421} C_VEL
LIN {X 0,Y 576.184,Z 621.684,A -85,B 0,C 180,E1 -9805.819,E2 -9805.819} C_VEL
LIN {X 0,Y 576.179,Z 625.334,A -85,B 0,C 180,E1 -9807.215,E2 -9807.215} C_VEL
LIN {X 0,Y 576.146,Z 627.519,A -85,B 0,C 180,E1 -9808.608,E2 -9808.608} C_VEL
LIN {X 0,Y 576.18,Z 628.293,A -85,B 0,C 180,E1 -9810.002,E2 -9810.002} C_VEL
LIN {X 0,Y 576.145,Z 627.655,A -85,B 0,C 180,E1 -9811.395,E2 -9811.395} C_VEL
LIN {X 0,Y 576.181,Z 625.582,A -85,B 0,C 180,E1 -9812.789,E2 -9812.789} C_VEL
LIN {X 0,Y 576.184,Z 622.046,A -85,B 0,C 180,E1 -9814.184,E2 -9814.184} C_VEL
LIN {X 0,Y 576.244,Z 616.953,A -85,B 0,C 180,E1 -9815.582,E2 -9815.582} C_VEL
LIN {X 0,Y 576.344,Z 612.008,A -85,B 0,C 180,E1 -9816.632,E2 -9816.632} C_VEL
LIN {X 0,Y 576.537,Z 604.851,A -85,B 0,C 180,E1 -9817.857,E2 -9817.857} C_VEL
LIN {X 0,Y 576.853,Z 595.961,A -85,B 0,C 180,E1 -9819.084,E2 -9819.084} C_VEL
LIN {X 0,Y 577.191,Z 586.638,A -85,B 0,C 180,E1 -9820.136,E2 -9820.136} C_VEL
LIN {X 0,Y 577.637,Z 575.266,A -85,B 0,C 180,E1 -9821.189,E2 -9821.189} C_VEL
LIN {X 0,Y 578.032,Z 563.68,A -85,B 0,C 180,E1 -9822.067,E2 -9822.067} C_VEL
LIN {X 0,Y 578.698,Z 549.371,A -85,B 0,C 180,E1 -9822.941,E2 -9822.941} C_VEL
LIN {X 0,Y 579.243,Z 536.212,A -85,B 0,C 180,E1 -9823.596,E2 -9823.596} C_VEL
LIN {X 0,Y 579.694,Z 522.523,A -85,B 0,C 180,E1 -9824.12,E2 -9824.12} C_VEL
LIN {X 0,Y 580.185,Z 508.342,A -85,B 0,C 180,E1 -9824.509,E2 -9824.509} C_VEL
LIN {X 0,Y 580.472,Z 493.767,A -85,B 0,C 180,E1 -9824.764,E2 -9824.764} C_VEL
LIN {X 0,Y 581.02,Z 423.302,A -85,B 0,C 180,E1 -9825.65,E2 -9825.65} C_VEL
LIN {X 0,Y 581.43,Z 387.571,A -85,B 0,C 180,E1 -9826.179,E2 -9826.179} C_VEL
LIN {X 0,Y 578.116,Z 360.2,A -85,B 0,C 180,E1 -9826.734,E2 -9826.734} C_VEL
LIN {X 0,Y 578.934,Z 335.663,A -85,B 0,C 180,E1 -9829.803,E2 -9829.803} C_VEL
LIN {X 0,Y 579.913,Z 312.387,A -85,B 0,C 180,E1 -9832.739,E2 -9832.739} C_VEL
LIN {X 0,Y 580.372,Z 300.727,A -85,B 0,C 180,E1 -9834.228,E2 -9834.228} C_VEL
LIN {X 0,Y 577.369,Z 285.127,A -85,B 0,C 180,E1 -9836.379,E2 -9836.379} C_VEL
LIN {X 0,Y 577.337,Z 285.126,A -85,B 0,C 180,E1 -9839.129,E2 -9839.129} C_VEL
LIN {X 0,Y 577.321,Z 285.126,A -85,B 0,C 180,E1 -9842.267,E2 -9842.267} C_VEL
LIN {X 0,Y 577.333,Z 285.126,A -85,B 0,C 180,E1 -9844.767,E2 -9844.767} C_VEL
LIN {X 0,Y 577.319,Z 285.132,A -85,B 0,C 180,E1 -9847.348,E2 -9847.348} C_VEL
LIN {X 0,Y 577.328,Z 285.126,A -85,B 0,C 180,E1 -9850.151,E2 -9850.151} C_VEL
LIN {X 0,Y 577.32,Z 285.132,A -85,B 0,C 180,E1 -9853.284,E2 -9853.284} C_VEL
LIN {X 0,Y 577.338,Z 285.124,A -85,B 0,C 180,E1 -9856.248,E2 -9856.248} C_VEL
LIN {X 0,Y 577.312,Z 285.134,A -85,B 0,C 180,E1 -9859.067,E2 -9859.067} C_VEL
LIN {X 0,Y 577.302,Z 285.129,A -85,B 0,C 180,E1 -9861.772,E2 -9861.772} C_VEL
LIN {X 0,Y 577.383,Z 285.122,A -85,B 0,C 180,E1 -9864.387,E2 -9864.387} C_VEL
LIN {X 0,Y 577.333,Z 285.129,A -85,B 0,C 180,E1 -9866.91,E2 -9866.91} C_VEL
LIN {X 0,Y 577.326,Z 285.126,A -85,B 0,C 180,E1 -9869.477,E2 -9869.477} C_VEL
LIN {X 0,Y 577.363,Z 285.128,A -85,B 0,C 180,E1 -9872.33,E2 -9872.33} C_VEL
LIN {X 0,Y 577.385,Z 285.122,A -85,B 0,C 180,E1 -9875.64,E2 -9875.64} C_VEL
LIN {X 0,Y 577.401,Z 285.124,A -85,B 0,C 180,E1 -9878.658,E2 -9878.658} C_VEL
LIN {X 0,Y 577.382,Z 285.126,A -85,B 0,C 180,E1 -9881.614,E2 -9881.614} C_VEL
LIN {X 0,Y 577.402,Z 285.12,A -85,B 0,C 180,E1 -9884.521,E2 -9884.521} C_VEL
LIN {X 0,Y 577.418,Z 285.12,A -85,B 0,C 180,E1 -9886.675,E2 -9886.675} C_VEL
LIN {X 0,Y 577.419,Z 285.266,A -85,B 0,C 180,E1 -9887.766,E2 -9887.766} C_VEL
LIN {X 0,Y 580.132,Z 298.352,A -85,B 0,C 180,E1 -9889.566,E2 -9889.566} C_VEL
LIN {X 0,Y 579.884,Z 316.656,A -85,B 0,C 180,E1 -9891.901,E2 -9891.901} C_VEL
LIN {X 0,Y 579.107,Z 342.882,A -85,B 0,C 180,E1 -9895.23,E2 -9895.23} C_VEL
LIN {X 0,Y 582.121,Z 359.737,A -85,B 0,C 180,E1 -9895.611,E2 -9895.611} C_VEL
LIN {X 0,Y 582.172,Z 368.821,A -85,B 0,C 180,E1 -9895.752,E2 -9895.752} C_VEL
LIN {X 0,Y 580.606,Z 481.955,A -85,B 0,C 180,E1 -9897.385,E2 -9897.385} C_VEL
LIN {X 0,Y 580.3,Z 495.491,A -85,B 0,C 180,E1 -9897.708,E2 -9897.708} C_VEL
LIN {X 0,Y 579.823,Z 509.51,A -85,B 0,C 180,E1 -9898.183,E2 -9898.183} C_VEL
LIN {X 0,Y 579.331,Z 522.895,A -85,B 0,C 180,E1 -9898.788,E2 -9898.788} C_VEL
LIN {X 0,Y 578.797,Z 535.085,A -85,B 0,C 180,E1 -9899.48,E2 -9899.48} C_VEL
LIN {X 0,Y 578.346,Z 547.397,A -85,B 0,C 180,E1 -9900.347,E2 -9900.347} C_VEL
LIN {X 0,Y 577.883,Z 557.577,A -85,B 0,C 180,E1 -9901.215,E2 -9901.215} C_VEL
LIN {X 0,Y 577.327,Z 567.777,A -85,B 0,C 180,E1 -9902.26,E2 -9902.26} C_VEL
LIN {X 0,Y 576.998,Z 576.195,A -85,B 0,C 180,E1 -9903.306,E2 -9903.306} C_VEL
LIN {X 0,Y 576.69,Z 583.218,A -85,B 0,C 180,E1 -9904.354,E2 -9904.354} C_VEL
LIN {X 0,Y 576.529,Z 589.94,A -85,B 0,C 180,E1 -9905.578,E2 -9905.578} C_VEL
LIN {X 0,Y 576.372,Z 594.561,A -85,B 0,C 180,E1 -9906.63,E2 -9906.63} C_VEL
LIN {X 0,Y 576.202,Z 598.277,A -85,B 0,C 180,E1 -9907.685,E2 -9907.685} C_VEL
LIN {X 0,Y 576.127,Z 601.873,A -85,B 0,C 180,E1 -9909.094,E2 -9909.094} C_VEL
LIN {X 0,Y 576.148,Z 603.458,A -85,B 0,C 180,E1 -9910.016,E2 -9910.016} C_VEL
LIN {X 0,Y 576.036,Z 604.568,A -85,B 0,C 180,E1 -9911.219,E2 -9911.219} C_VEL
LIN {X 0,Y 576.061,Z 604.579,A -85,B 0,C 180,E1 -9912.642,E2 -9912.642} C_VEL
LIN {X 0,Y 576.132,Z 603.936,A -85,B 0,C 180,E1 -9913.436,E2 -9913.436} C_VEL
LIN {X 0,Y 576.069,Z 601.829,A -85,B 0,C 180,E1 -9914.794,E2 -9914.794} C_VEL
LIN {X 0,Y 576.188,Z 598.105,A -85,B 0,C 180,E1 -9916.236,E2 -9916.236} C_VEL
LIN {X 0,Y 576.28,Z 594.211,A -85,B 0,C 180,E1 -9917.325,E2 -9917.325} C_VEL
LIN {X 0,Y 576.459,Z 588.352,A -85,B 0,C 180,E1 -9918.599,E2 -9918.599} C_VEL
LIN {X 0,Y 576.7,Z 580.874,A -85,B 0,C 180,E1 -9919.882,E2 -9919.882} C_VEL
LIN {X 0,Y 577.021,Z 572.547,A -85,B 0,C 180,E1 -9921.036,E2 -9921.036} C_VEL
LIN {X 0,Y 577.37,Z 563.287,A -85,B 0,C 180,E1 -9922.091,E2 -9922.091} C_VEL
LIN {X 0,Y 577.789,Z 552.869,A -85,B 0,C 180,E1 -9923.072,E2 -9923.072} C_VEL
LIN {X 0,Y 578.258,Z 541.711,A -85,B 0,C 180,E1 -9923.94,E2 -9923.94} C_VEL
LIN {X 0,Y 578.688,Z 529.41,A -85,B 0,C 180,E1 -9924.726,E2 -9924.726} C_VEL
LIN {X 0,Y 579.18,Z 515.67,A -85,B 0,C 180,E1 -9925.425,E2 -9925.425} C_VEL
LIN {X 0,Y 579.616,Z 501.336,A -85,B 0,C 180,E1 -9925.981,E2 -9925.981} C_VEL
LIN {X 0,Y 580.038,Z 487.308,A -85,B 0,C 180,E1 -9926.37,E2 -9926.37} C_VEL
LIN {X 0,Y 580.211,Z 472.308,A -85,B 0,C 180,E1 -9926.642,E2 -9926.642} C_VEL
LIN {X 0,Y 581.356,Z 359.801,A -85,B 0,C 180,E1 -9928.181,E2 -9928.181} C_VEL
LIN {X 0,Y 578.583,Z 342.086,A -85,B 0,C 180,E1 -9928.52,E2 -9928.52} C_VEL
LIN {X 0,Y 579.195,Z 318.811,A -85,B 0,C 180,E1 -9931.536,E2 -9931.536} C_VEL
LIN {X 0,Y 579.726,Z 298.409,A -85,B 0,C 180,E1 -9934.182,E2 -9934.182} C_VEL
LIN {X 0,Y 577.688,Z 286.489,A -85,B 0,C 180,E1 -9935.818,E2 -9935.818} C_VEL
LIN {X 0,Y 577.414,Z 285.121,A -85,B 0,C 180,E1 -9936.022,E2 -9936.022} C_VEL
LIN {X 0,Y 577.318,Z 285.126,A -85,B 0,C 180,E1 -9939.117,E2 -9939.117} C_VEL
LIN {X 0,Y 577.35,Z 285.129,A -85,B 0,C 180,E1 -9942.262,E2 -9942.262} C_VEL
LIN {X 0,Y 577.365,Z 285.122,A -85,B 0,C 180,E1 -9945.279,E2 -9945.279} C_VEL
LIN {X 0,Y 577.308,Z 285.133,A -85,B 0,C 180,E1 -9948.139,E2 -9948.139} C_VEL
LIN {X 0,Y 577.319,Z 285.129,A -85,B 0,C 180,E1 -9950.941,E2 -9950.941} C_VEL
LIN {X 0,Y 577.315,Z 285.13,A -85,B 0,C 180,E1 -9953.521,E2 -9953.521} C_VEL
LIN {X 0,Y 577.318,Z 285.129,A -85,B 0,C 180,E1 -9956.074,E2 -9956.074} C_VEL
LIN {X 0,Y 577.307,Z 285.13,A -85,B 0,C 180,E1 -9959.015,E2 -9959.015} C_VEL
LIN {X 0,Y 576.641,Z 285.216,A -85,B 0,C 180,E1 -9959.598,E2 -9959.598} C_VEL
LIN {X 0,Y 573.779,Z 285.572,A -85,B 0,C 180,E1 -9960.543,E2 -9960.543} C_VEL
LIN {X 0,Y 571.375,Z 285.87,A -85,B 0,C 180,E1 -9961.303,E2 -9961.303} C_VEL
LIN {X 0,Y 570.364,Z 285.995,A -85,B 0,C 180,E1 -9961.89,E2 -9961.89} C_VEL
LIN {X 0,Y 570.293,Z 286.004,A -85,B 0,C 180,E1 -9962.089,E2 -9962.089} C_VEL
LIN {X 0,Y 570.271,Z 286.01,A -85,B 0,C 180,E1 -9964.538,E2 -9964.538} C_VEL
LIN {X 0,Y 570.323,Z 286,A -85,B 0,C 180,E1 -9967.09,E2 -9967.09} C_VEL
LIN {X 0,Y 570.325,Z 286,A -85,B 0,C 180,E1 -9969.885,E2 -9969.885} C_VEL
LIN {X 0,Y 570.347,Z 285.996,A -85,B 0,C 180,E1 -9972.856,E2 -9972.856} C_VEL
LIN {X 0,Y 570.395,Z 285.994,A -85,B 0,C 180,E1 -9975.958,E2 -9975.958} C_VEL
LIN {X 0,Y 570.419,Z 285.986,A -85,B 0,C 180,E1 -9979.222,E2 -9979.222} C_VEL
LIN {X 0,Y 570.449,Z 285.988,A -85,B 0,C 180,E1 -9982.236,E2 -9982.236} C_VEL
LIN {X 0,Y 570.478,Z 286.136,A -85,B 0,C 180,E1 -9982.99,E2 -9982.99} C_VEL
LIN {X 0,Y 571.567,Z 293.621,A -85,B 0,C 180,E1 -9984.372,E2 -9984.372} C_VEL
LIN {X 0,Y 571.433,Z 299.763,A -85,B 0,C 180,E1 -9985.453,E2 -9985.453} C_VEL
LIN {X 0,Y 574.644,Z 315.513,A -85,B 0,C 180,E1 -9985.739,E2 -9985.739} C_VEL
LIN {X 0,Y 573.719,Z 434.673,A -85,B 0,C 180,E1 -9987.243,E2 -9987.243} C_VEL
LIN {X 0,Y 573.44,Z 449.308,A -85,B 0,C 180,E1 -9987.57,E2 -9987.57} C_VEL
LIN {X 0,Y 573.108,Z 463.185,A -85,B 0,C 180,E1 -9988.028,E2 -9988.028} C_VEL
LIN {X 0,Y 572.745,Z 476.068,A -85,B 0,C 180,E1 -9988.597,E2 -9988.597} C_VEL
LIN {X 0,Y 572.312,Z 488.564,A -85,B 0,C 180,E1 -9989.297,E2 -9989.297} C_VEL
LIN {X 0,Y 571.674,Z 500.025,A -85,B 0,C 180,E1 -9990.086,E2 -9990.086} C_VEL
LIN {X 0,Y 571.258,Z 511.443,A -85,B 0,C 180,E1 -9991.052,E2 -9991.052} C_VEL
LIN {X 0,Y 570.67,Z 521.72,A -85,B 0,C 180,E1 -9992.108,E2 -9992.108} C_VEL
LIN {X 0,Y 570.321,Z 530.184,A -85,B 0,C 180,E1 -9993.166,E2 -9993.166} C_VEL
LIN {X 0,Y 569.862,Z 538.327,A -85,B 0,C 180,E1 -9994.404,E2 -9994.404} C_VEL
LIN {X 0,Y 569.733,Z 544.857,A -85,B 0,C 180,E1 -9995.643,E2 -9995.643} C_VEL
LIN {X 0,Y 569.477,Z 550.689,A -85,B 0,C 180,E1 -9997.063,E2 -9997.063} C_VEL
LIN {X 0,Y 569.255,Z 554.97,A -85,B 0,C 180,E1 -9998.489,E2 -9998.489} C_VEL
LIN {X 0,Y 569.228,Z 557.805,A -85,B 0,C 180,E1 -9999.918,E2 -9999.918} C_VEL
LIN {X 0,Y 569.143,Z 559.285,A -85,B 0,C 180,E1 -10001.354,E2 -10001.354} C_VEL
LIN {X 0,Y 569.187,Z 559.411,A -85,B 0,C 180,E1 -10002.796,E2 -10002.796} C_VEL
LIN {X 0,Y 569.22,Z 558.171,A -85,B 0,C 180,E1 -10004.245,E2 -10004.245} C_VEL
LIN {X 0,Y 569.355,Z 555.495,A -85,B 0,C 180,E1 -10005.701,E2 -10005.701} C_VEL
LIN {X 0,Y 569.545,Z 551.307,A -85,B 0,C 180,E1 -10007.165,E2 -10007.165} C_VEL
LIN {X 0,Y 569.802,Z 547.112,A -85,B 0,C 180,E1 -10008.266,E2 -10008.266} C_VEL
LIN {X 0,Y 570.104,Z 540.863,A -85,B 0,C 180,E1 -10009.558,E2 -10009.558} C_VEL
LIN {X 0,Y 570.586,Z 532.975,A -85,B 0,C 180,E1 -10010.853,E2 -10010.853} C_VEL
LIN {X 0,Y 571.065,Z 524.651,A -85,B 0,C 180,E1 -10011.966,E2 -10011.966} C_VEL
LIN {X 0,Y 571.657,Z 514.511,A -85,B 0,C 180,E1 -10013.082,E2 -10013.082} C_VEL
LIN {X 0,Y 572.25,Z 504.239,A -85,B 0,C 180,E1 -10014.013,E2 -10014.013} C_VEL
LIN {X 0,Y 572.891,Z 492.045,A -85,B 0,C 180,E1 -10014.922,E2 -10014.922} C_VEL
LIN {X 0,Y 573.387,Z 480.804,A -85,B 0,C 180,E1 -10015.601,E2 -10015.601} C_VEL
LIN {X 0,Y 573.894,Z 468.299,A -85,B 0,C 180,E1 -10016.208,E2 -10016.208} C_VEL
LIN {X 0,Y 574.36,Z 454.424,A -85,B 0,C 180,E1 -10016.722,E2 -10016.722} C_VEL
LIN {X 0,Y 574.604,Z 440.711,A -85,B 0,C 180,E1 -10017.084,E2 -10017.084} C_VEL
LIN {X 0,Y 574.744,Z 425.234,A -85,B 0,C 180,E1 -10017.336,E2 -10017.336} C_VEL
LIN {X 0,Y 575.709,Z 315.966,A -85,B 0,C 180,E1 -10018.721,E2 -10018.721} C_VEL
LIN {X 0,Y 572.101,Z 300.065,A -85,B 0,C 180,E1 -10019.076,E2 -10019.076} C_VEL
LIN {X 0,Y 572.114,Z 295.897,A -85,B 0,C 180,E1 -10019.837,E2 -10019.837} C_VEL
LIN {X 0,Y 570.307,Z 286.005,A -85,B 0,C 180,E1 -10021.772,E2 -10021.772} C_VEL
LIN {X 0,Y 570.268,Z 286.008,A -85,B 0,C 180,E1 -10024.619,E2 -10024.619} C_VEL
LIN {X 0,Y 570.267,Z 286.005,A -85,B 0,C 180,E1 -10027.024,E2 -10027.024} C_VEL
LIN {X 0,Y 570.263,Z 286.007,A -85,B 0,C 180,E1 -10029.692,E2 -10029.692} C_VEL
LIN {X 0,Y 570.277,Z 286.007,A -85,B 0,C 180,E1 -10032.528,E2 -10032.528} C_VEL
LIN {X 0,Y 570.293,Z 285.996,A -85,B 0,C 180,E1 -10035.566,E2 -10035.566} C_VEL
LIN {X 0,Y 570.265,Z 286.006,A -85,B 0,C 180,E1 -10038.522,E2 -10038.522} C_VEL
LIN {X 0,Y 570.255,Z 286.006,A -85,B 0,C 180,E1 -10041.213,E2 -10041.213} C_VEL
LIN {X 0,Y 570.326,Z 285.986,A -85,B 0,C 180,E1 -10044.148,E2 -10044.148} C_VEL
LIN {X 0,Y 570.258,Z 286.004,A -85,B 0,C 180,E1 -10046.636,E2 -10046.636} C_VEL
LIN {X 0,Y 570.294,Z 286.001,A -85,B 0,C 180,E1 -10049.284,E2 -10049.284} C_VEL
LIN {X 0,Y 570.305,Z 285.996,A -85,B 0,C 180,E1 -10052.179,E2 -10052.179} C_VEL
LIN {X 0,Y 570.293,Z 286.006,A -85,B 0,C 180,E1 -10055.345,E2 -10055.345} C_VEL
LIN {X 0,Y 570.298,Z 286.004,A -85,B 0,C 180,E1 -10057.62,E2 -10057.62} C_VEL
LIN {X 0,Y 570.295,Z 286,A -85,B 0,C 180,E1 -10059.885,E2 -10059.885} C_VEL
LIN {X 0,Y 570.294,Z 286,A -85,B 0,C 180,E1 -10062.118,E2 -10062.118} C_VEL
LIN {X 0,Y 570.374,Z 285.993,A -85,B 0,C 180,E1 -10065.055,E2 -10065.055} C_VEL
LIN {X 0,Y 570.354,Z 285.994,A -85,B 0,C 180,E1 -10067.949,E2 -10067.949} C_VEL
LIN {X 0,Y 570.362,Z 285.987,A -85,B 0,C 180,E1 -10070.1,E2 -10070.1} C_VEL
LIN {X 0,Y 570.42,Z 285.986,A -85,B 0,C 180,E1 -10072.947,E2 -10072.947} C_VEL
LIN {X 0,Y 570.468,Z 285.972,A -85,B 0,C 180,E1 -10075.775,E2 -10075.775} C_VEL
LIN {X 0,Y 570.636,Z 285.963,A -85,B 0,C 180,E1 -10079.297,E2 -10079.297} C_VEL
LIN {X 0,Y 570.537,Z 285.965,A -85,B 0,C 180,E1 -10081.407,E2 -10081.407} C_VEL
LIN {X 0,Y 570.5,Z 285.982,A -85,B 0,C 180,E1 -10084.93,E2 -10084.93} C_VEL
LIN {X 0,Y 570.425,Z 285.977,A -85,B 0,C 180,E1 -10087.763,E2 -10087.763} C_VEL
LIN {X 0,Y 570.438,Z 285.988,A -85,B 0,C 180,E1 -10090.802,E2 -10090.802} C_VEL
LIN {X 0,Y 570.378,Z 285.987,A -85,B 0,C 180,E1 -10094.218,E2 -10094.218} C_VEL
LIN {X 0,Y 570.332,Z 285.991,A -85,B 0,C 180,E1 -10097.143,E2 -10097.143} C_VEL
LIN {X 0,Y 570.299,Z 285.999,A -85,B 0,C 180,E1 -10099.367,E2 -10099.367} C_VEL
LIN {X 0,Y 570.31,Z 285.993,A -85,B 0,C 180,E1 -10101.62,E2 -10101.62} C_VEL
LIN {X 0,Y 570.311,Z 285.997,A -85,B 0,C 180,E1 -10103.91,E2 -10103.91} C_VEL
LIN {X 0,Y 570.266,Z 286.005,A -85,B 0,C 180,E1 -10107.03,E2 -10107.03} C_VEL
LIN {X 0,Y 570.292,Z 285.999,A -85,B 0,C 180,E1 -10109.425,E2 -10109.425} C_VEL
LIN {X 0,Y 570.301,Z 286.002,A -85,B 0,C 180,E1 -10112.068,E2 -10112.068} C_VEL
LIN {X 0,Y 570.324,Z 285.98,A -85,B 0,C 180,E1 -10115.256,E2 -10115.256} C_VEL
LIN {X 0,Y 570.319,Z 285.995,A -85,B 0,C 180,E1 -10117.885,E2 -10117.885} C_VEL
LIN {X 0,Y 570.288,Z 286.006,A -85,B 0,C 180,E1 -10120.614,E2 -10120.614} C_VEL
LIN {X 0,Y 570.277,Z 286.002,A -85,B 0,C 180,E1 -10123.562,E2 -10123.562} C_VEL
LIN {X 0,Y 570.286,Z 286.004,A -85,B 0,C 180,E1 -10126.546,E2 -10126.546} C_VEL
LIN {X 0,Y 570.294,Z 286,A -85,B 0,C 180,E1 -10129.389,E2 -10129.389} C_VEL
LIN {X 0,Y 570.324,Z 286.006,A -85,B 0,C 180,E1 -10132.118,E2 -10132.118} C_VEL
LIN {X 0,Y 570.331,Z 286.002,A -85,B 0,C 180,E1 -10134.747,E2 -10134.747} C_VEL
LIN {X 0,Y 570.287,Z 286.007,A -85,B 0,C 180,E1 -10137.29,E2 -10137.29} C_VEL
LIN {X 0,Y 570.294,Z 286.011,A -85,B 0,C 180,E1 -10139.766,E2 -10139.766} C_VEL
LIN {X 0,Y 570.327,Z 286.063,A -85,B 0,C 180,E1 -10142.778,E2 -10142.778} C_VEL
LIN {X 0,Y 573.956,Z 302.994,A -85,B 0,C 180,E1 -10145.298,E2 -10145.298} C_VEL
LIN {X 0,Y 574.054,Z 307.217,A -85,B 0,C 180,E1 -10145.875,E2 -10145.875} C_VEL
LIN {X 0,Y 572.918,Z 326.981,A -85,B 0,C 180,E1 -10148.485,E2 -10148.485} C_VEL
LIN {X 0,Y 571.825,Z 349.628,A -85,B 0,C 180,E1 -10151.431,E2 -10151.431} C_VEL
LIN {X 0,Y 571.332,Z 361.448,A -85,B 0,C 180,E1 -10152.954,E2 -10152.954} C_VEL
LIN {X 0,Y 574.798,Z 385.2,A -85,B 0,C 180,E1 -10153.384,E2 -10153.384} C_VEL
LIN {X 0,Y 575.314,Z 390.932,A -85,B 0,C 180,E1 -10153.475,E2 -10153.475} C_VEL
LIN {X 0,Y 574.274,Z 499.476,A -85,B 0,C 180,E1 -10154.86,E2 -10154.86} C_VEL
LIN {X 0,Y 573.807,Z 513.617,A -85,B 0,C 180,E1 -10155.171,E2 -10155.171} C_VEL
LIN {X 0,Y 573.262,Z 527.712,A -85,B 0,C 180,E1 -10155.632,E2 -10155.632} C_VEL
LIN {X 0,Y 572.624,Z 540.798,A -85,B 0,C 180,E1 -10156.202,E2 -10156.202} C_VEL
LIN {X 0,Y 571.953,Z 553.47,A -85,B 0,C 180,E1 -10156.907,E2 -10156.907} C_VEL
LIN {X 0,Y 571.302,Z 565.031,A -85,B 0,C 180,E1 -10157.702,E2 -10157.702} C_VEL
LIN {X 0,Y 570.695,Z 576.642,A -85,B 0,C 180,E1 -10158.677,E2 -10158.677} C_VEL
LIN {X 0,Y 570.227,Z 587.06,A -85,B 0,C 180,E1 -10159.742,E2 -10159.742} C_VEL
LIN {X 0,Y 569.783,Z 595.677,A -85,B 0,C 180,E1 -10160.806,E2 -10160.806} C_VEL
LIN {X 0,Y 569.433,Z 603.967,A -85,B 0,C 180,E1 -10162.048,E2 -10162.048} C_VEL
LIN {X 0,Y 569.213,Z 612.902,A -85,B 0,C 180,E1 -10163.643,E2 -10163.643} C_VEL
LIN {X 0,Y 569.15,Z 617.656,A -85,B 0,C 180,E1 -10164.706,E2 -10164.706} C_VEL
LIN {X 0,Y 569.09,Z 621.457,A -85,B 0,C 180,E1 -10165.767,E2 -10165.767} C_VEL
LIN {X 0,Y 569.104,Z 625.136,A -85,B 0,C 180,E1 -10167.18,E2 -10167.18} C_VEL
LIN {X 0,Y 569.052,Z 627.345,A -85,B 0,C 180,E1 -10168.591,E2 -10168.591} C_VEL
LIN {X 0,Y 569.083,Z 628.139,A -85,B 0,C 180,E1 -10170.002,E2 -10170.002} C_VEL
LIN {X 0,Y 569.051,Z 627.524,A -85,B 0,C 180,E1 -10171.412,E2 -10171.412} C_VEL
LIN {X 0,Y 569.106,Z 625.472,A -85,B 0,C 180,E1 -10172.824,E2 -10172.824} C_VEL
LIN {X 0,Y 569.093,Z 621.948,A -85,B 0,C 180,E1 -10174.237,E2 -10174.237} C_VEL
LIN {X 0,Y 569.154,Z 618.32,A -85,B 0,C 180,E1 -10175.298,E2 -10175.298} C_VEL
LIN {X 0,Y 569.219,Z 613.69,A -85,B 0,C 180,E1 -10176.36,E2 -10176.36} C_VEL
LIN {X 0,Y 569.384,Z 607.004,A -85,B 0,C 180,E1 -10177.601,E2 -10177.601} C_VEL
LIN {X 0,Y 569.685,Z 598.67,A -85,B 0,C 180,E1 -10178.842,E2 -10178.842} C_VEL
LIN {X 0,Y 569.976,Z 589.921,A -85,B 0,C 180,E1 -10179.908,E2 -10179.908} C_VEL
LIN {X 0,Y 570.49,Z 579.307,A -85,B 0,C 180,E1 -10180.972,E2 -10180.972} C_VEL
LIN {X 0,Y 570.902,Z 568.594,A -85,B 0,C 180,E1 -10181.861,E2 -10181.861} C_VEL
LIN {X 0,Y 571.388,Z 556.927,A -85,B 0,C 180,E1 -10182.659,E2 -10182.659} C_VEL
LIN {X 0,Y 571.944,Z 544.145,A -85,B 0,C 180,E1 -10183.367,E2 -10183.367} C_VEL
LIN {X 0,Y 572.556,Z 528.815,A -85,B 0,C 180,E1 -10184.029,E2 -10184.029} C_VEL
LIN {X 0,Y 572.998,Z 516.341,A -85,B 0,C 180,E1 -10184.446,E2 -10184.446} C_VEL
LIN {X 0,Y 573.385,Z 502.45,A -85,B 0,C 180,E1 -10184.776,E2 -10184.776} C_VEL
LIN {X 0,Y 573.693,Z 479.069,A -85,B 0,C 180,E1 -10185.098,E2 -10185.098} C_VEL
LIN {X 0,Y 573.973,Z 443.124,A -85,B 0,C 180,E1 -10185.575,E2 -10185.575} C_VEL
LIN {X 0,Y 574.729,Z 388.251,A -85,B 0,C 180,E1 -10186.399,E2 -10186.399} C_VEL
LIN {X 0,Y 571.493,Z 361.881,A -85,B 0,C 180,E1 -10186.937,E2 -10186.937} C_VEL
LIN {X 0,Y 571.07,Z 359.025,A -85,B 0,C 180,E1 -10187.017,E2 -10187.017} C_VEL
LIN {X 0,Y 571.919,Z 336.636,A -85,B 0,C 180,E1 -10189.851,E2 -10189.851} C_VEL
LIN {X 0,Y 572.959,Z 313.231,A -85,B 0,C 180,E1 -10192.841,E2 -10192.841} C_VEL
LIN {X 0,Y 573.376,Z 301.563,A -85,B 0,C 180,E1 -10194.351,E2 -10194.351} C_VEL
LIN {X 0,Y 570.329,Z 286.003,A -85,B 0,C 180,E1 -10196.536,E2 -10196.536} C_VEL
LIN {X 0,Y 570.296,Z 286.005,A -85,B 0,C 180,E1 -10199.426,E2 -10199.426} C_VEL
LIN {X 0,Y 570.28,Z 286.004,A -85,B 0,C 180,E1 -10202.06,E2 -10202.06} C_VEL
LIN {X 0,Y 570.285,Z 286.004,A -85,B 0,C 180,E1 -10204.622,E2 -10204.622} C_VEL
LIN {X 0,Y 570.28,Z 286.006,A -85,B 0,C 180,E1 -10207.026,E2 -10207.026} C_VEL
LIN {X 0,Y 570.282,Z 286.008,A -85,B 0,C 180,E1 -10209.695,E2 -10209.695} C_VEL
LIN {X 0,Y 570.263,Z 286.004,A -85,B 0,C 180,E1 -10212.526,E2 -10212.526} C_VEL
LIN {X 0,Y 570.31,Z 286.003,A -85,B 0,C 180,E1 -10215.568,E2 -10215.568} C_VEL
LIN {X 0,Y 570.271,Z 286.006,A -85,B 0,C 180,E1 -10218.526,E2 -10218.526} C_VEL
LIN {X 0,Y 570.268,Z 286.009,A -85,B 0,C 180,E1 -10221.214,E2 -10221.214} C_VEL
LIN {X 0,Y 570.33,Z 285.999,A -85,B 0,C 180,E1 -10224.153,E2 -10224.153} C_VEL
LIN {X 0,Y 570.283,Z 286.009,A -85,B 0,C 180,E1 -10226.639,E2 -10226.639} C_VEL
LIN {X 0,Y 570.293,Z 286.003,A -85,B 0,C 180,E1 -10229.291,E2 -10229.291} C_VEL
LIN {X 0,Y 570.335,Z 286.001,A -85,B 0,C 180,E1 -10232.18,E2 -10232.18} C_VEL
LIN {X 0,Y 570.322,Z 286.001,A -85,B 0,C 180,E1 -10235.347,E2 -10235.347} C_VEL
LIN {X 0,Y 570.34,Z 286.007,A -85,B 0,C 180,E1 -10238.381,E2 -10238.381} C_VEL
LIN {X 0,Y 570.339,Z 286.003,A -85,B 0,C 180,E1 -10241.379,E2 -10241.379} C_VEL
LIN {X 0,Y 570.345,Z 286.001,A -85,B 0,C 180,E1 -10244.325,E2 -10244.325} C_VEL
LIN {X 0,Y 570.386,Z 285.997,A -85,B 0,C 180,E1 -10246.507,E2 -10246.507} C_VEL
LIN {X 0,Y 570.376,Z 286.064,A -85,B 0,C 180,E1 -10247.522,E2 -10247.522} C_VEL
LIN {X 0,Y 573.302,Z 299.875,A -85,B 0,C 180,E1 -10249.44,E2 -10249.44} C_VEL
LIN {X 0,Y 573.058,Z 317.917,A -85,B 0,C 180,E1 -10251.76,E2 -10251.76} C_VEL
LIN {X 0,Y 572.276,Z 343.39,A -85,B 0,C 180,E1 -10254.997,E2 -10254.997} C_VEL
